(* IEC 61131-3 sources: elnaProjects/ElpcLogic/PomarKc7Changed/FunctionBlocks (part 7) *)

(* ---- proc_IM_Init.st ---- *)
FUNCTION_BLOCK proc_IM_Init

VAR_INPUT
	init : BOOL; (*Флаг необходимости инициализации структур-дескрипторов.*)
END_VAR

VAR
	stKr_Ini : fb_Kran_Init; (*ФБ инициализации кранов*)
	stSw_Ini : fb_Switch_Init; (*ФБ инициализации Switchs*)
	stOp_Ini : fb_OilPump_Init; (*ФБ инициализации НУ*)
	stSSw_Ini : fb_SectionSwitch_Init; (*ФБ инициализации МВ*)
	stAp_Ini : fb_AnalogParametr_Init; (*ФБ инициализации Аналогового параметра*)
	stDp_Ini : fb_DiscretParametr_Init; (*ФБ инициализации Дискретного параметра*)
	stSs_Ini : fb_singleSignal_Init; (*ФБ инициализации singleSignal*)
	stSo_Ini : fb_singleOutput_Init; (*ФБ инициализации singleOutput*)
	inits : UINT; (*Текущее количество успешно проинициализированных структур-дескрипторов.*)
END_VAR

VAR_INPUT
	initiales : UINT; (*Общее количество успешно проинициализированных структур-дескрипторов.*)
END_VAR

VAR_EXTERNAL
	IM : ImConfig;
END_VAR

inits := 0; (* Флаг необходимости инициализации структур-дескрипторов *)
                                     (* Стартовая инициализация ИМ *)
(* Кран 1 *)
stKr_Ini(data_Ini := true, ISVALIDREF_statOn:=true, ISVALIDREF_statOff:=true,
      ISVALIDREF_cmdOn:=true, ISVALIDREF_cmdOff:=true,
      ISVALIDREF_inSo:=true, ISVALIDREF_inSz:=true,
      str_Kr := IM.Kran1);
inits := inits + BOOL_TO_UINT(stKr_Ini.Init);

(* Кран 2 *)
stKr_Ini(data_Ini := true, ISVALIDREF_statOn:=true, ISVALIDREF_statOff:=true,
      ISVALIDREF_cmdOn:=true, ISVALIDREF_cmdOff:=true,
      ISVALIDREF_inSo:=true, ISVALIDREF_inSz:=true,
      str_Kr := IM.Kran2);
inits := inits + BOOL_TO_UINT(stKr_Ini.Init);

(* Кран 3 *)
stKr_Ini(data_Ini := true, ISVALIDREF_statOn:=true, ISVALIDREF_statOff:=true,
      ISVALIDREF_cmdOn:=true, ISVALIDREF_cmdOff:=true,
      ISVALIDREF_inSo:=true, ISVALIDREF_inSz:=true,
      str_Kr := IM.Kran3);
inits := inits + BOOL_TO_UINT(stKr_Ini.Init);

(* Кран 3b *)
stKr_Ini(data_Ini := true, ISVALIDREF_statOn:=true, ISVALIDREF_statOff:=true,
      ISVALIDREF_cmdOn:=true, ISVALIDREF_cmdOff:=true,
      ISVALIDREF_inSo:=true, ISVALIDREF_inSz:=true,
      str_Kr := IM.Kran3b);
inits := inits + BOOL_TO_UINT(stKr_Ini.Init);

(* Кран 4 *)
stKr_Ini(data_Ini := true, ISVALIDREF_statOn:=true, ISVALIDREF_statOff:=true,
      ISVALIDREF_cmdOn:=true, ISVALIDREF_cmdOff:=true,
      ISVALIDREF_inSo:=true, ISVALIDREF_inSz:=true,
      str_Kr := IM.Kran4);
inits := inits + BOOL_TO_UINT(stKr_Ini.Init);

(* Кран 5 *)
stKr_Ini(data_Ini := true, ISVALIDREF_statOn:=true, ISVALIDREF_statOff:=true,
      ISVALIDREF_cmdOn:=true, ISVALIDREF_cmdOff:=true,
      ISVALIDREF_inSo:=true, ISVALIDREF_inSz:=true, continueHoldCommand:=T#5S,
      str_Kr := IM.Kran5);
inits := inits + BOOL_TO_UINT(stKr_Ini.Init);

(* Кран 6 *)
stKr_Ini(data_Ini := true, ISVALIDREF_statOn:=true, ISVALIDREF_statOff:=true,
      ISVALIDREF_cmdOn:=true, ISVALIDREF_cmdOff:=true,
      str_Kr := IM.Kran6);
inits := inits + BOOL_TO_UINT(stKr_Ini.Init);

(* НУ1 Насос уплотнения *)
stOp_Ini(data_Ini := true, ISVALIDREF_statOn:=true, ISVALIDREF_statOff:=true,
      ISVALIDREF_cmdOn:=true, ISVALIDREF_cmdOff:=true,
      str_Op := IM.nu1);
inits := inits + BOOL_TO_UINT(stOp_Ini.Init);

(* НУ2 Насос уплотнения *)
stOp_Ini(data_Ini := true, ISVALIDREF_statOn:=true, ISVALIDREF_statOff:=true,
      ISVALIDREF_cmdOn:=true, ISVALIDREF_cmdOff:=true,
      str_Op := IM.nu2);
inits := inits + BOOL_TO_UINT(stOp_Ini.Init);

(* ПНС Насос смазки *)
stSw_Ini(data_Ini := true, ISVALIDREF_statOn:=true, ISVALIDREF_statOff:=true,
      ISVALIDREF_cmdOn:=true, ISVALIDREF_cmdOff:=true,
      str_Sw := IM.pns);
inits := inits + BOOL_TO_UINT(stSw_Ini.Init);

(* В1 АВОМ вентилятор охлаждения *)
stSw_Ini(data_Ini := true, ISVALIDREF_statOn:=true, ISVALIDREF_statOff:=true,
      ISVALIDREF_cmdOn:=true, ISVALIDREF_cmdOff:=true,
      str_Sw := IM.v1_Avom);
inits := inits + BOOL_TO_UINT(stSw_Ini.Init);

(* В2 АВОМ вентилятор охлаждения *)
stSw_Ini(data_Ini := true, ISVALIDREF_statOn:=true, ISVALIDREF_statOff:=true,
      ISVALIDREF_cmdOn:=true, ISVALIDREF_cmdOff:=true,
      str_Sw := IM.v2_Avom);
inits := inits + BOOL_TO_UINT(stSw_Ini.Init);

(* В3 АВОМ вентилятор охлаждения *)
stSw_Ini(data_Ini := true, ISVALIDREF_statOn:=true, ISVALIDREF_statOff:=true,
      ISVALIDREF_cmdOn:=true, ISVALIDREF_cmdOff:=true,
      str_Sw := IM.v3_Avom);
inits := inits + BOOL_TO_UINT(stSw_Ini.Init);

(* В4 АВОМ вентилятор охлаждения *)
stSw_Ini(data_Ini := true, ISVALIDREF_statOn:=true, ISVALIDREF_statOff:=true,
      ISVALIDREF_cmdOn:=true, ISVALIDREF_cmdOff:=true,
      str_Sw := IM.v4_Avom);
inits := inits + BOOL_TO_UINT(stSw_Ini.Init);

(* МВ масляный выключатель *)
stSSw_Ini(data_Ini := true, ISVALIDREF_statOn:=true, ISVALIDREF_statOff:=true,
      ISVALIDREF_cmdOn:=true, ISVALIDREF_cmdOff:=true,
      ISVALIDREF_basketRolledIn:=true, ISVALIDREF_basketRolledout:=true,
      str_Sw := IM.mv);
inits := inits + BOOL_TO_UINT(stSSw_Ini.Init);

(* В4 АВОМ вентилятор охлаждения *)
stSw_Ini(data_Ini := true, ISVALIDREF_statOn:=true, ISVALIDREF_statOff:=true,
      ISVALIDREF_cmdOn:=true, ISVALIDREF_cmdOff:=true,
      str_Sw := IM.KaloriferAVOM);
inits := inits + BOOL_TO_UINT(stSw_Ini.Init);

(* В4 АВОМ вентилятор охлаждения *)
stSw_Ini(data_Ini := true, ISVALIDREF_statOn:=true, ISVALIDREF_statOff:=true,
      ISVALIDREF_cmdOn:=true, ISVALIDREF_cmdOff:=true,
      str_Sw := IM.CMN);
inits := inits + BOOL_TO_UINT(stSw_Ini.Init);

(* В4 АВОМ вентилятор охлаждения *)
stSw_Ini(data_Ini := true, ISVALIDREF_statOn:=true, ISVALIDREF_statOff:=true,
      ISVALIDREF_cmdOn:=true, ISVALIDREF_cmdOff:=true,
      str_Sw := IM.TEN_kollectora);
inits := inits + BOOL_TO_UINT(stSw_Ini.Init);

(* В4 АВОМ вентилятор охлаждения *)
stSw_Ini(data_Ini := true, ISVALIDREF_statOn:=true, ISVALIDREF_statOff:=true,
      ISVALIDREF_cmdOn:=true, ISVALIDREF_cmdOff:=true,
      str_Sw := IM.TEN_MB);
inits := inits + BOOL_TO_UINT(stSw_Ini.Init);

                                     (* Стартовая инициализация singleSignal *)
    (* Перепад давления «газ-газ» на кране 1 ≤1 кгс/см² *)
stSs_Ini(data_Ini := true, inverse:=FALSE, (*DelayOn:=T#0S, DelayOff:=T#0S,*) str_SS := IM.SingleSignals.dP_maslo_gaz_Less100);
inits := inits + BOOL_TO_UINT(stSs_Ini.Init);

 (* Осевой сдвиг ротора вправо ≥3,7 кгс/см² *)
stSs_Ini(data_Ini := true, inverse:=FALSE, (*DelayOn:=T#0S, DelayOff:=T#0S,*) str_SS := IM.SingleSignals.dp_kran1_Less100);
inits := inits + BOOL_TO_UINT(stSs_Ini.Init);

    (* Пробой вентиля *)
stSs_Ini(data_Ini := true, inverse:=TRUE, (*DelayOn:=T#0S, DelayOff:=T#0S,*) str_SS := IM.SingleSignals.Vozbud_neispr_tsepey_upr_AVR_pit);
inits := inits + BOOL_TO_UINT(stSs_Ini.Init);

    (* Работа схемы ресинхронизации *)
stSs_Ini(data_Ini := true, inverse:=FALSE, (*DelayOn:=T#0S, DelayOff:=T#0S,*) str_SS := IM.SingleSignals.Vozbud_gotovnost);
inits := inits + BOOL_TO_UINT(stSs_Ini.Init);

    (* Контроль состояния возбудительного устройства  *)
stSs_Ini(data_Ini := true, inverse:=FALSE, (*DelayOn:=T#0S, DelayOff:=T#0S,*) str_SS := IM.SingleSignals.Vozbud_neispravnost);
inits := inits + BOOL_TO_UINT(stSs_Ini.Init);

    (* Неисправность форсировки воз-буждения  *)
stSs_Ini(data_Ini := true, inverse:=FALSE, (*DelayOn:=T#0S, DelayOff:=T#0S,*) str_SS := IM.SingleSignals.SHAVR1_v_rabote);
inits := inits + BOOL_TO_UINT(stSs_Ini.Init);

  (* Неисправность возбудительного устройства  *)
stSs_Ini(data_Ini := true, inverse:=FALSE, (*DelayOn:=T#0S, DelayOff:=T#0S,*) str_SS := IM.SingleSignals.SHAVR2_v_rabote);
inits := inits + BOOL_TO_UINT(stSs_Ini.Init);

  (* Готовность включения БЭО по отказу контроллера  *)
stSs_Ini(data_Ini := true, inverse:=FALSE, (*DelayOn:=T#0S, DelayOff:=T#0S,*) str_SS := IM.SingleSignals.Avariinoe_otkluch_vikluchatelya);
inits := inits + BOOL_TO_UINT(stSs_Ini.Init);

  (* Срабатывание БЭАО  *)
stSs_Ini(data_Ini := true, inverse:=FALSE, (*DelayOn:=T#0S, DelayOff:=T#0S,*) str_SS := IM.SingleSignals.Assinhronnii_hod_peregruzka);
inits := inits + BOOL_TO_UINT(stSs_Ini.Init);

  (* Выключатель основного ввода питания QF1  в положении включен   *)
stSs_Ini(data_Ini := true, inverse:=TRUE, (*DelayOn:=T#0S, DelayOff:=T#0S,*) str_SS := IM.SingleSignals.QF1_on);
inits := inits + BOOL_TO_UINT(stSs_Ini.Init);

  (* Выключатель резервного ввода питания QF2  в положении включен   *)
stSs_Ini(data_Ini := true, inverse:=TRUE, (*DelayOn:=T#0S, DelayOff:=T#0S,*) str_SS := IM.SingleSignals.QF2_on);
inits := inits + BOOL_TO_UINT(stSs_Ini.Init);

  (* Выключатель питания кранов:  QF23 110 В в положении включен   *)
stSs_Ini(data_Ini := true, inverse:=TRUE, (*DelayOn:=T#0S, DelayOff:=T#0S,*) str_SS := IM.SingleSignals.QF23_on);
inits := inits + BOOL_TO_UINT(stSs_Ini.Init);

  (* Выключатели группы 1: QF4, QF5 в положении включен   *)
stSs_Ini(data_Ini := true, inverse:=TRUE, (*DelayOn:=T#0S, DelayOff:=T#0S,*) str_SS := IM.SingleSignals.QF4_QF5_on);
inits := inits + BOOL_TO_UINT(stSs_Ini.Init);

  (* Выключатели группы 2: QF6, QF7 в положении включен   *)
stSs_Ini(data_Ini := true, inverse:=TRUE, (*DelayOn:=T#0S, DelayOff:=T#0S,*) str_SS := IM.SingleSignals.QF6_QF7_on);
inits := inits + BOOL_TO_UINT(stSs_Ini.Init);

  (* Выключатели группы 3: QF8, QF9 в положении включен   *)
stSs_Ini(data_Ini := true, inverse:=TRUE, (*DelayOn:=T#0S, DelayOff:=T#0S,*) str_SS := IM.SingleSignals.QF8_QF9_on);
inits := inits + BOOL_TO_UINT(stSs_Ini.Init);

  (* Выключатели группы 4: QF10, QF11 в положении включен   *)
stSs_Ini(data_Ini := true, inverse:=TRUE, (*DelayOn:=T#0S, DelayOff:=T#0S,*) str_SS := IM.SingleSignals.QF10_QF11_on);
inits := inits + BOOL_TO_UINT(stSs_Ini.Init);

  (* Выключатели группы 5: QF12, QF13 в положении включен   *)
stSs_Ini(data_Ini := true, inverse:=TRUE, (*DelayOn:=T#0S, DelayOff:=T#0S,*) str_SS := IM.SingleSignals.QF12_QF13_on);
inits := inits + BOOL_TO_UINT(stSs_Ini.Init);

  (* Выключатели группы 6: QF14, QF15 в положении включен   *)
stSs_Ini(data_Ini := true, inverse:=TRUE, (*DelayOn:=T#0S, DelayOff:=T#0S,*) str_SS := IM.SingleSignals.QF14_QF15_on);
inits := inits + BOOL_TO_UINT(stSs_Ini.Init);

  (* Выключатели группы : QF22 в положении включен   *)
stSs_Ini(data_Ini := true, inverse:=TRUE, (*DelayOn:=T#0S, DelayOff:=T#0S,*) str_SS := IM.SingleSignals.QF22_on);
inits := inits + BOOL_TO_UINT(stSs_Ini.Init);

  (* Неисправность источников питания группы 1: G1, G2 (=24 В)   *)
stSs_Ini(data_Ini := true, inverse:=TRUE, (*DelayOn:=T#0S, DelayOff:=T#0S,*) str_SS := IM.SingleSignals.NS_G1_G2);
inits := inits + BOOL_TO_UINT(stSs_Ini.Init);

  (* Неисправность источников питания группы 2: G3, G4 (=24 В)   *)
stSs_Ini(data_Ini := true, inverse:=TRUE, (*DelayOn:=T#0S, DelayOff:=T#0S,*) str_SS := IM.SingleSignals.NS_G3_G4);
inits := inits + BOOL_TO_UINT(stSs_Ini.Init);

  (* Неисправность источников питания внутренних ПТС: G15, G16 (=24 В)   *)
stSs_Ini(data_Ini := true, inverse:=TRUE, (*DelayOn:=T#0S, DelayOff:=T#0S,*) str_SS := IM.SingleSignals.NS_G15_G16);
inits := inits + BOOL_TO_UINT(stSs_Ini.Init);

  (* Неисправность источника питания аналоговых сигналов: G17 (=24 В)   *)
stSs_Ini(data_Ini := true, inverse:=TRUE, (*DelayOn:=T#0S, DelayOff:=T#0S,*) str_SS := IM.SingleSignals.NS_G17);
inits := inits + BOOL_TO_UINT(stSs_Ini.Init);

  (* Неисправность источников питания группы 3: G5, G6 (=24 В)   *)
stSs_Ini(data_Ini := true, inverse:=TRUE, (*DelayOn:=T#0S, DelayOff:=T#0S,*) str_SS := IM.SingleSignals.NS_G5_G6);
inits := inits + BOOL_TO_UINT(stSs_Ini.Init);

  (* Неисправность источников питания группы 4: G7, G8 (=24 В)   *)
stSs_Ini(data_Ini := true, inverse:=TRUE, (*DelayOn:=T#0S, DelayOff:=T#0S,*) str_SS := IM.SingleSignals.NS_G7_G8);
inits := inits + BOOL_TO_UINT(stSs_Ini.Init);

  (* Неисправность источников питания внешних цепей: G18, G19 (=24 В)   *)
stSs_Ini(data_Ini := true, inverse:=TRUE, (*DelayOn:=T#0S, DelayOff:=T#0S,*) str_SS := IM.SingleSignals.NS_G18_G19);
inits := inits + BOOL_TO_UINT(stSs_Ini.Init);

  (* Неисправность источников питания группы 5: G9, G10, G11, G12 (=110 В)   *)
stSs_Ini(data_Ini := true, inverse:=TRUE, (*DelayOn:=T#0S, DelayOff:=T#0S,*) str_SS := IM.SingleSignals.NS_G10_G11);
inits := inits + BOOL_TO_UINT(stSs_Ini.Init);

  (* Неисправность источников питания G13, G14 (=24 В)   *)
stSs_Ini(data_Ini := true, inverse:=TRUE, (*DelayOn:=T#0S, DelayOff:=T#0S,*) str_SS := IM.SingleSignals.NS_G13_G14);
inits := inits + BOOL_TO_UINT(stSs_Ini.Init);

    (* Неисправность источников питания G13, G14 (=24 В)   *)
stSs_Ini(data_Ini := true, inverse:=TRUE, (*DelayOn:=T#0S, DelayOff:=T#0S,*) str_SS := IM.SingleSignals.Uroven_masla_akkum);
inits := inits + BOOL_TO_UINT(stSs_Ini.Init);

  (* Неисправность источников питания G13, G14 (=24 В)   *)
stSs_Ini(data_Ini := true, inverse:=TRUE, (*DelayOn:=T#0S, DelayOff:=T#0S,*) str_SS := IM.SingleSignals.BEAO_srabotal);
inits := inits + BOOL_TO_UINT(stSs_Ini.Init);

  (* Неисправность источников питания G13, G14 (=24 В)   *)
stSs_Ini(data_Ini := true, inverse:=TRUE, (*DelayOn:=T#0S, DelayOff:=T#0S,*) str_SS := IM.SingleSignals.Chastotny_pusk);
inits := inits + BOOL_TO_UINT(stSs_Ini.Init);

  (* Неисправность источников питания G13, G14 (=24 В)   *)
stSs_Ini(data_Ini := true, inverse:=TRUE, (*DelayOn:=T#0S, DelayOff:=T#0S,*) str_SS := IM.SingleSignals.Neuspesh_chastotny_pusk);
inits := inits + BOOL_TO_UINT(stSs_Ini.Init);

  (* Неисправность источников питания G13, G14 (=24 В)   *)
stSs_Ini(data_Ini := true, inverse:=TRUE, (*DelayOn:=T#0S, DelayOff:=T#0S,*) str_SS := IM.SingleSignals.Rezhim_ruchnogo_regulirovaniya);
inits := inits + BOOL_TO_UINT(stSs_Ini.Init);

  (* Неисправность источников питания G13, G14 (=24 В)   *)
stSs_Ini(data_Ini := true, inverse:=TRUE, (*DelayOn:=T#0S, DelayOff:=T#0S,*) str_SS := IM.SingleSignals.SHU_v_GPA_vkluch);
inits := inits + BOOL_TO_UINT(stSs_Ini.Init);

  (* Неисправность источников питания G13, G14 (=24 В)   *)
stSs_Ini(data_Ini := true, inverse:=TRUE, (*DelayOn:=T#0S, DelayOff:=T#0S,*) str_SS := IM.SingleSignals.SHP_v_GPA_vkluch);
inits := inits + BOOL_TO_UINT(stSs_Ini.Init);

(* Отключение МВ1 от КНА   *)
stSs_Ini(data_Ini := true, inverse:=TRUE, (*wait_time:=T#0S,*) str_SS := IM.SingleSignals.NKU1_GPA_on);
inits := inits + BOOL_TO_UINT(stSs_Ini.Init);

(* Отключение МВ1 от КНА   *)
stSs_Ini(data_Ini := true, inverse:=TRUE, (*wait_time:=T#0S,*) str_SS := IM.SingleSignals.NKU2_GPA_on);
inits := inits + BOOL_TO_UINT(stSs_Ini.Init);

(* Отключение МВ1 от КНА   *)
stSs_Ini(data_Ini := true, inverse:=TRUE, (*wait_time:=T#0S,*) str_SS := IM.SingleSignals.AO_KC_ot_SHKS);
inits := inits + BOOL_TO_UINT(stSs_Ini.Init);

(* Отключение МВ1 от КНА   *)
stSs_Ini(data_Ini := true, inverse:=TRUE, (*wait_time:=T#0S,*) str_SS := IM.SingleSignals.AO_GPA_ot_SHU);
inits := inits + BOOL_TO_UINT(stSs_Ini.Init);

(* Отключение МВ1 от КНА   *)
stSs_Ini(data_Ini := true, inverse:=TRUE, (*wait_time:=T#0S,*) str_SS := IM.SingleSignals.Razreshenie_zagruzki_dvig);
inits := inits + BOOL_TO_UINT(stSs_Ini.Init);

(* Отключение МВ1 от КНА   *)
stSs_Ini(data_Ini := true, inverse:=TRUE, (*wait_time:=T#0S,*) str_SS := IM.SingleSignals.Osnovnoy_regul_off);
inits := inits + BOOL_TO_UINT(stSs_Ini.Init);

(* Отключение МВ1 от КНА   *)
stSs_Ini(data_Ini := true, inverse:=TRUE, (*wait_time:=T#0S,*) str_SS := IM.SingleSignals.Voltage_sekcii_norm);
inits := inits + BOOL_TO_UINT(stSs_Ini.Init);

(* Отключение МВ1 от КНА   *)
stSs_Ini(data_Ini := true, inverse:=TRUE, (*wait_time:=T#0S,*) str_SS := IM.SingleSignals.Reactorny_pusk);
inits := inits + BOOL_TO_UINT(stSs_Ini.Init);

(* Отключение МВ1 от КНА   *)
stSs_Ini(data_Ini := true, inverse:=TRUE, (*wait_time:=T#0S,*) str_SS := IM.SingleSignals.NO_GPA_ot_SHU);
inits := inits + BOOL_TO_UINT(stSs_Ini.Init);

(* Отключение МВ1 от КНА   *)
stSs_Ini(data_Ini := true, inverse:=TRUE, (*wait_time:=T#0S,*) str_SS := IM.SingleSignals.AO_GPA_ot_PRU);
inits := inits + BOOL_TO_UINT(stSs_Ini.Init);

(* Отключение МВ1 от КНА   *)
stSs_Ini(data_Ini := true, inverse:=TRUE, (*wait_time:=T#0S,*) str_SS := IM.SingleSignals.Nalichie_BP1);
inits := inits + BOOL_TO_UINT(stSs_Ini.Init);

(* Отключение МВ1 от КНА   *)
stSs_Ini(data_Ini := true, inverse:=TRUE, (*wait_time:=T#0S,*) str_SS := IM.SingleSignals.Nalichie_BP2);
inits := inits + BOOL_TO_UINT(stSs_Ini.Init);

(* Отключение МВ1 от КНА   *)
stSs_Ini(data_Ini := true, inverse:=TRUE, (*wait_time:=T#0S,*) str_SS := IM.SingleSignals.Nalichie_BP3);
inits := inits + BOOL_TO_UINT(stSs_Ini.Init);

(* Отключение МВ1 от КНА   *)
stSs_Ini(data_Ini := true, inverse:=TRUE, (*wait_time:=T#0S,*) str_SS := IM.SingleSignals.Nalichie_BP4);
inits := inits + BOOL_TO_UINT(stSs_Ini.Init);

(* Отключение МВ1 от КНА   *)
stSs_Ini(data_Ini := true, inverse:=TRUE, (*wait_time:=T#0S,*) str_SS := IM.SingleSignals.Nalichie_BP5);
inits := inits + BOOL_TO_UINT(stSs_Ini.Init);

(* Отключение МВ1 от КНА   *)
stSs_Ini(data_Ini := true, inverse:=TRUE, (*wait_time:=T#0S,*) str_SS := IM.SingleSignals.Nalichie_BP6);
inits := inits + BOOL_TO_UINT(stSs_Ini.Init);

(* Отключение МВ1 от КНА   *)
stSs_Ini(data_Ini := true, inverse:=TRUE, (*wait_time:=T#0S,*) str_SS := IM.SingleSignals.Nalichie_BP7_BP8);
inits := inits + BOOL_TO_UINT(stSs_Ini.Init);

(* Отключение МВ1 от КНА   *)
stSs_Ini(data_Ini := true, inverse:=TRUE, (*wait_time:=T#0S,*) str_SS := IM.SingleSignals.Nalichie_BP9_BP10);
inits := inits + BOOL_TO_UINT(stSs_Ini.Init);

(* Отключение МВ1 от КНА   *)
stSs_Ini(data_Ini := true, inverse:=TRUE, (*wait_time:=T#0S,*) str_SS := IM.SingleSignals.Nalichie_cepei_upravlen_mv);
inits := inits + BOOL_TO_UINT(stSs_Ini.Init);

(* Отключение МВ1 от КНА   *)
stSs_Ini(data_Ini := true, inverse:=TRUE, (*wait_time:=T#0S,*) str_SS := IM.SingleSignals.Nalichie_220BEAO);
inits := inits + BOOL_TO_UINT(stSs_Ini.Init);

(* Отключение МВ1 от КНА   *)
stSs_Ini(data_Ini := true, inverse:=TRUE, (*wait_time:=T#0S,*) str_SS := IM.SingleSignals.Nalichie_per_220_na_vhode);
inits := inits + BOOL_TO_UINT(stSs_Ini.Init);

(* Отключение МВ1 от КНА   *)
stSs_Ini(data_Ini := true, inverse:=TRUE, (*wait_time:=T#0S,*) str_SS := IM.SingleSignals.Nalichie_post_220_na_vhode);
inits := inits + BOOL_TO_UINT(stSs_Ini.Init);

(* Отключение МВ1 от КНА   *)
stSs_Ini(data_Ini := true, inverse:=TRUE, (*wait_time:=T#0S,*) str_SS := IM.SingleSignals.Nalichie_BP11);
inits := inits + BOOL_TO_UINT(stSs_Ini.Init);

(* Отключение МВ1 от КНА   *)
stSs_Ini(data_Ini := true, inverse:=TRUE, (*wait_time:=T#0S,*) str_SS := IM.SingleSignals.Nalichie_BP12);
inits := inits + BOOL_TO_UINT(stSs_Ini.Init);

(* Отключение МВ1 от КНА   *)
stSs_Ini(data_Ini := true, inverse:=TRUE, (*wait_time:=T#0S,*) str_SS := IM.SingleSignals.Dver_SHU_pered_otkrita);
inits := inits + BOOL_TO_UINT(stSs_Ini.Init);

(* Отключение МВ1 от КНА   *)
stSs_Ini(data_Ini := true, inverse:=TRUE, (*wait_time:=T#0S,*) str_SS := IM.SingleSignals.Dver_SHU_zad_otkrita);
inits := inits + BOOL_TO_UINT(stSs_Ini.Init);

(* Отключение МВ1 от КНА   *)
stSs_Ini(data_Ini := true, inverse:=TRUE, (*wait_time:=T#0S,*) str_SS := IM.SingleSignals.EO_GPA_ot_knopki_SHU);
inits := inits + BOOL_TO_UINT(stSs_Ini.Init);

(* Отключение МВ1 от КНА   *)
stSs_Ini(data_Ini := true, inverse:=TRUE, (*wait_time:=T#0S,*) str_SS := IM.SingleSignals.EO_EGPA_ot_PRY);
inits := inits + BOOL_TO_UINT(stSs_Ini.Init);

(* Отключение МВ1 от КНА   *)
stSs_Ini(data_Ini := true, inverse:=TRUE, (*wait_time:=T#0S,*) str_SS := IM.SingleSignals.Synchroniz_rezhima_K1);
inits := inits + BOOL_TO_UINT(stSs_Ini.Init);

                                     (* Стартовая инициализация singleOutput *)
(* Идикация НО (подсветка кнопки на шкафу)   *)
stSo_Ini(data_Ini := true, inOpcCommandsDisabled:=TRUE, (*wait_time:=T#0S,*) str_SO := IM.SingleOutputs.Rabota_EGPA);
inits := inits + BOOL_TO_UINT(stSo_Ini.Init);

(* Взвод включения БЭАО по неисправности ПТС   *)
stSo_Ini(data_Ini := true, inOpcCommandsDisabled:=TRUE, wait_time:=T#0S, str_SO := IM.SingleOutputs.Neispr_EGPA);
inits := inits + BOOL_TO_UINT(stSo_Ini.Init);

(* Авария ЭГПА в КЦ   *)
stSo_Ini(data_Ini := true, inOpcCommandsDisabled:=TRUE, (*wait_time:=T#0S,*) str_SO := IM.SingleOutputs.Avary_EGPA);
inits := inits + BOOL_TO_UINT(stSo_Ini.Init);

(* Авария ЭГПА в КЦ   *)
stSo_Ini(data_Ini := true, inOpcCommandsDisabled:=TRUE, (*wait_time:=T#0S,*) str_SO := IM.SingleOutputs.U_lamp_SHU);
inits := inits + BOOL_TO_UINT(stSo_Ini.Init);

(* Индикация ПС Фонарь   *)
stSo_Ini(data_Ini := true, inOpcCommandsDisabled:=TRUE, (*wait_time:=T#0S,*) str_SO := IM.SingleOutputs.AO_knopka_ind);
inits := inits + BOOL_TO_UINT(stSo_Ini.Init);

(* Индикация АС Фонарь   *)
stSo_Ini(data_Ini := true, inOpcCommandsDisabled:=TRUE, (*wait_time:=T#0S,*) str_SO := IM.SingleOutputs.Pusk_SHUP);
inits := inits + BOOL_TO_UINT(stSo_Ini.Init);

(* Отключение МВ1 от КНА   *)
stSo_Ini(data_Ini := true, inOpcCommandsDisabled:=TRUE, (*wait_time:=T#0S,*) str_SO := IM.SingleOutputs.Stop_SHUP);
inits := inits + BOOL_TO_UINT(stSo_Ini.Init);

(* Отключение МВ1 от КНА   *)
stSo_Ini(data_Ini := true, inOpcCommandsDisabled:=TRUE, (*wait_time:=T#0S,*) str_SO := IM.SingleOutputs.NO_fonar);
inits := inits + BOOL_TO_UINT(stSo_Ini.Init);

(* Отключение МВ1 от КНА   *)
stSo_Ini(data_Ini := true, inOpcCommandsDisabled:=TRUE, (*wait_time:=T#0S,*) str_SO := IM.SingleOutputs.PC_fonar);
inits := inits + BOOL_TO_UINT(stSo_Ini.Init);

(* Отключение МВ1 от КНА   *)
stSo_Ini(data_Ini := true, inOpcCommandsDisabled:=TRUE, (*wait_time:=T#0S,*) str_SO := IM.SingleOutputs.AC_fonar);
inits := inits + BOOL_TO_UINT(stSo_Ini.Init);

(* Отключение МВ1 от КНА   *)
stSo_Ini(data_Ini := true, inOpcCommandsDisabled:=TRUE, (*wait_time:=T#0S,*) str_SO := IM.SingleOutputs.Kr1_smazka);
inits := inits + BOOL_TO_UINT(stSo_Ini.Init);

(* Отключение МВ1 от КНА   *)
stSo_Ini(data_Ini := true, inOpcCommandsDisabled:=TRUE, (*wait_time:=T#0S,*) str_SO := IM.SingleOutputs.Kr2_smazka);
inits := inits + BOOL_TO_UINT(stSo_Ini.Init);

(* Отключение МВ1 от КНА   *)
stSo_Ini(data_Ini := true, inOpcCommandsDisabled:=TRUE, (*wait_time:=T#0S,*) str_SO := IM.SingleOutputs.Kr4_open_from_alg);
inits := inits + BOOL_TO_UINT(stSo_Ini.Init);

(* Отключение МВ1 от КНА   *)
stSo_Ini(data_Ini := true, inOpcCommandsDisabled:=TRUE, (*wait_time:=T#0S,*) str_SO := IM.SingleOutputs.Synch_rej_K1);
inits := inits + BOOL_TO_UINT(stSo_Ini.Init);
initiales := 0;

IF init THEN initiales := inits; END_IF;

(* ---- proc_Protection.st ---- *)
FUNCTION_BLOCK proc_Protection

VAR
	fb_mvOff : fb_MvProtection;
	fb_dPmaslo_gaz_Less100 : fb_DiProtection; (*[A1-14:1, AI0] Резерв*)
	fb_Reg_vozb_off : fb_DiProtection; (*[A1-14:2, AI1] Резерв*)
	fb_Fail_chastotnii_pusk : fb_DiProtection;
	fb_Off_avar_vikluchatel : fb_DiProtection;
	fb_AOKC_SHKC : fb_DiProtection;
	fb_AO_PRU : fb_DiProtection;
	fb_AO_ot_SHU : fb_DiProtection;
	fb_Kran1_sdvig : fb_KranOpenProtection;
	fb_Kran2_sdvig : fb_KranOpenProtection;
	fb_Toporno_podshipnika_EDT_1 : fb_AiProtection;
	fb_Toy_podshipnika_EDT_2 : fb_AiProtection;
	fb_Toy_podshipnika_kol_EDT_3 : fb_AiProtection;
	fb_Toy_podshipnika_kol_EDT_4 : fb_AiProtection;
	fb_Toy_podshipnika_shest_red_EDT_5 : fb_AiProtection;
	fb_Ty_podshipnika_red_EDT_6 : fb_AiProtection;
	fb_Ty_podshipnika_nagnet_EDT_7_1 : fb_AiProtection;
	fb_Ty_podshipnika_nagnet_EDT_7_2 : fb_AiProtection;
	fb_Toy_podshipnika_svobod_konca_EDT_8_1 : fb_AiProtection;
	fb_Toy_podshipnika_svobod_konca_EDT_8_2 : fb_AiProtection;
	fb_Toy_podshipnika_rab_kol_EDT_9_1 : fb_AiProtection;
	fb_Toy_podshipnika_rab_kol_EDT_9_2 : fb_AiProtection;
	fb_Toy_podshipnika_nerab_kol_EDT_10_1 : fb_AiProtection;
	fb_Toy_podshipnika_nerab_kol_EDT_10_2 : fb_AiProtection;
	fb_Tgaza_na_vhode_H : fb_AiProtection;
	fb_Tgaza_na_vyhode_H : fb_AiProtection;
	fb_Tmasla_v_mb : fb_AiProtection;
	fb_Tmasla_v_mb_nad_ten : fb_AiProtection;
	fb_Tgorjachego_vozduha_ED_kanal_1 : fb_AiProtection;
	fb_Tgorjachego_vozduha_ED_kanal_2 : fb_AiProtection;
	fb_Tmasla_do_AVOM : fb_AiProtection;
	fb_Tmasla_posle_AVOM : fb_AiProtection;
	fb_Tmedi_statora_kanal_1 : fb_AiProtection;
	fb_Tmedi_statora_kanal_2 : fb_AiProtection;
	fb_Tmedi_statora_kanal_3 : fb_AiProtection;
	fb_Tstali_statora_kanal_1 : fb_AiProtection;
	fb_Tstali_statora_kanal_2 : fb_AiProtection;
	fb_Tstali_statora_kanal_3 : fb_AiProtection;
	fb_Tholodnogo_vozduha_ED_kanal_1 : fb_AiProtection;
	fb_Tholodnogo_vozduha_ED_kanal_2 : fb_AiProtection;
	fb_Pmaslo_sm_nizkoe : fb_AiProtection;
	fb_Pmaslo_sm_vysokoe : fb_AiProtection;
	fb_Pgaza_na_vhode_nagnetatelia : fb_AiProtection;
	fb_Pgaza_na_vyhode_nagnetatelia : fb_AiProtection;
	fb_Pmasla_posle_NU : fb_AiProtection;
	fb_Pmasla_smazki_posle_gns : fb_AiProtection;
	fb_Pimpuls_gaz : fb_AiProtection;
	fb_dPmaslo_gaz : fb_AiProtection;
	fb_dP_maslo_na_filtre : fb_AiProtection;
	fb_Os_sdvig_nagnetatelja_plus : fb_AiProtection;
	fb_Os_sdvig_nagnetatelja_minus : fb_AiProtection;
	fb_Vibro_skorost_OPED_T1 : fb_AiProtection;
	fb_Vibro_skorost_OPED_T2 : fb_AiProtection;
	fb_Vibro_skorost_OYP_kolesa_ED_T3 : fb_AiProtection;
	fb_Vibro_skorost_OP_kolesa_RH_T4 : fb_AiProtection;
	fb_Vibro_skorost_OP_shesterni_RED_T5 : fb_AiProtection;
	fb_Vibro_skorost_OP_shesterni_RED_T6 : fb_AiProtection;
	fb_Vibroperemesh_vala_N_T7 : fb_AiProtection;
	fb_Vibroperemesh_vala_N_T8 : fb_AiProtection;
	fb_Uroven_masla_v_mb : fb_AiProtection;
	fb_Tok_statora : fb_AiProtection;
	fb_Kontrol_per_220V_less187 : fb_AiProtection;
	fb_Kontrol_per_220V_high242 : fb_AiProtection;
	fb_Kontrol_post_220V_less187 : fb_AiProtection;
	fb_Kontrol_post_220V_high242 : fb_AiProtection;
END_VAR

VAR_EXTERNAL
	protections : ProtectionsConfig;
	ai : AiConfig;
	IM : ImConfig;
END_VAR

(************************************************************* DiProtection ************************************************************)
(* МВ отключен
fb_mvOff(sw:=IM.mv, StrDIp := protections.Pgaza_na_vyhode_nagnetatelia_GPA_STOP);*)

(* Неисправность возбудительного устройства *)
fb_dPmaslo_gaz_Less100(di := IM.SingleSignals.dP_maslo_gaz_Less100, StrDIp := protections.dPmaslo_gaz_less100);

(* Сдвиг крана №2 *)
fb_Reg_vozb_off(di:=IM.SingleSignals.Vozbud_neispravnost, StrDIp := protections.Reg_vozb_off);

(* Сдвиг крана №2 *)
fb_Fail_chastotnii_pusk(di:=IM.SingleSignals.Neuspesh_chastotny_pusk, StrDIp := protections.Fail_chastotnii_pusk);

(* Сдвиг крана №2 *)
fb_Off_avar_vikluchatel(di:=IM.SingleSignals.Avariinoe_otkluch_vikluchatelya, StrDIp := protections.Off_avar_vikluchatel);

(* Сдвиг крана №2 *)
fb_AOKC_SHKC(di:=IM.SingleSignals.AO_KC_ot_SHKS, StrDIp := protections.AOKC_SHKC);

(* Сдвиг крана №2 *)
fb_AO_PRU(di:=IM.SingleSignals.AO_GPA_ot_PRU, StrDIp := protections.AO_PRU);

(* Сдвиг крана №2 *)
fb_AO_ot_SHU(di:=IM.SingleSignals.AO_GPA_ot_SHU, StrDIp := protections.AO_ot_SHU);

(* Сдвиг крана №2 *)
fb_Kran1_sdvig(im:=IM.Kran1, StrDIp := protections.Kran1_sdvig);

(* Сдвиг крана №2 *)
fb_Kran2_sdvig(im:=IM.Kran2, StrDIp := protections.Kran2_sdvig);

(************************************************************* AiProtection ************************************************************)

(* Температура переднего опорного подшипника двигателя, т.1 *)
fb_Toporno_podshipnika_EDT_1(ai := ai.Toporno_podshipnika_EDT_1, StrAIp := protections.Topornogo_podshipnika_EDT_1);

(* Температура заднего опорного подшипника двигателя, т.2 *)
fb_Toy_podshipnika_EDT_2(ai := ai.Toy_podshipnika_EDT_2, StrAIp := protections.Toy_podshipnika_EDT_2);

(* Температура подшипника редуктора, т1 *)
fb_Toy_podshipnika_kol_EDT_3(ai := ai.Toy_podshipnika_kol_EDT_3, StrAIp := protections.Toy_podshipnika_kol_EDT_3);

(* Температура подшипника редуктора, т2 *)
fb_Toy_podshipnika_kol_EDT_4(ai := ai.Toy_podshipnika_kol_EDT_4, StrAIp := protections.Toy_podshipnika_kol_EDT_4);

(* Температура подшипника редуктора, т3 *)
fb_Toy_podshipnika_shest_red_EDT_5(ai := ai.Toy_podshipnika_shest_red_EDT_5, StrAIp := protections.To_podshipnika_shest_red_EDT_5);

(* Температура подшипника редуктора, т4 *)
fb_Ty_podshipnika_red_EDT_6(ai := ai.Ty_podshipnika_red_EDT_6, StrAIp := protections.To_podshipnika_shest_red_EDT_6);

(* Температура опорного подшипника нагнетателя, т1 *)
fb_Ty_podshipnika_nagnet_EDT_7_1(ai := ai.Ty_podshipnika_nagnet_EDT_7_1, StrAIp := protections.To_podshipnika_N_EDT_7);

(* Температура опорного подшипника нагнетателя, т1 *)
fb_Ty_podshipnika_nagnet_EDT_7_2(ai := ai.Ty_podshipnika_nagnet_EDT_7_2, StrAIp := protections.To_podshipnika_N_EDT_7);

(* Температура опорного подшипника нагнетателя, т2 *)
fb_Toy_podshipnika_svobod_konca_EDT_8_1(ai := ai.Toy_podshipnika_svobod_konca_EDT_8_1, StrAIp := protections.To_podshipnika_svob_konca_EDT_8);

(* Температура опорного подшипника нагнетателя, т2 *)
fb_Toy_podshipnika_svobod_konca_EDT_8_2(ai := ai.Toy_podshipnika_svobod_konca_EDT_8_2, StrAIp := protections.To_podshipnika_svob_konca_EDT_8);

(* Температура опорного подшипника нагнетателя, т3 *)
fb_Toy_podshipnika_rab_kol_EDT_9_1(ai := ai.Toy_podshipnika_rab_kol_EDT_9_1, StrAIp := protections.Ty_podshipnika_rab_kol_EDT_9);

(* Температура опорного подшипника нагнетателя, т3 *)
fb_Toy_podshipnika_rab_kol_EDT_9_2(ai := ai.Toy_podshipnika_rab_kol_EDT_9_2, StrAIp := protections.Ty_podshipnika_rab_kol_EDT_9);

(* Температура упорно опорного подшипника нагнетателя, т4 *)
fb_Toy_podshipnika_nerab_kol_EDT_10_1(ai := ai.Toy_podshipnika_nerab_kol_EDT_10_1, StrAIp := protections.Typornogo_podshipnika_nerab_kolodok_HT_10);

(* Температура упорно опорного подшипника нагнетателя, т4 *)
fb_Toy_podshipnika_nerab_kol_EDT_10_2(ai := ai.Toy_podshipnika_nerab_kol_EDT_10_2, StrAIp := protections.Typornogo_podshipnika_nerab_kolodok_HT_10);

(* Температура газа на выходе нагнетателя *)
fb_Tgaza_na_vyhode_H(ai := ai.Tgaza_na_vhode_H, StrAIp := protections.Tgaza_na_vyhode_H);

(* Температура газа на выходе нагнетателя *)
fb_Os_sdvig_nagnetatelja_plus(ai := ai.Os_sdvig_nagnetatelja_plus, StrAIp := protections.Os_sdvig_nagnetatelja_plus);

(* Температура газа на выходе нагнетателя *)
fb_Os_sdvig_nagnetatelja_minus(ai := ai.Os_sdvig_nagnetatelja_minus, StrAIp := protections.Os_sdvig_nagnetatelja_minus);

(* Температура газа на выходе нагнетателя *)
fb_Pgaza_na_vyhode_nagnetatelia(ai := ai.Pgaza_na_vyhode_nagnetatelia, StrAIp := protections.Pgaza_na_vyhode_nagnetatelia);

(* Температура газа на выходе нагнетателя *)
fb_dPmaslo_gaz(ai := ai.dPmaslo_gaz, StrAIp := protections.dPmaslo_gaz);

(* Температура газа на выходе нагнетателя *)
fb_Pmaslo_sm_nizkoe(ai := ai.Pmaslo_sm_nizkoe, StrAIp := protections.Pmaslo_sm_nizkoe);

(* Температура газа на выходе нагнетателя *)
fb_Pmaslo_sm_vysokoe(ai := ai.Pmaslo_sm_vysokoe, StrAIp := protections.Pmaslo_sm_vysokoe);

(* Температура газа на выходе нагнетателя *)
fb_Vibro_skorost_OPED_T1(ai := ai.Vibro_skorost_OPED_T1, StrAIp := protections.Vibro_skorost_OPED_T1);

(* Температура газа на выходе нагнетателя *)
fb_Vibro_skorost_OPED_T2(ai := ai.Vibro_skorost_OYPED_T2, StrAIp := protections.Vibro_skorost_OPED_T2);

(* Температура газа на выходе нагнетателя *)
fb_Vibro_skorost_OYP_kolesa_ED_T3(ai := ai.Vibro_skorost_OYP_kolesa_ED_T3, StrAIp := protections.Vibro_skorost_OYP_kolesa_ED_T3);

(* Температура газа на выходе нагнетателя *)
fb_Vibro_skorost_OP_kolesa_RH_T4(ai := ai.Vibro_skorost_OP_kolesa_RH_T4, StrAIp := protections.Vibro_skorost_OP_kolesa_RH_T4);

(* Температура газа на выходе нагнетателя *)
fb_Vibro_skorost_OP_shesterni_RED_T5(ai := ai.Vibro_skorost_OP_shesterni_RED_T5, StrAIp := protections.Vibro_skorost_OP_shesterni_RED_T5);

(* Температура газа на выходе нагнетателя *)
fb_Vibro_skorost_OP_shesterni_RED_T6(ai := ai.Vibro_skorost_OP_shesterni_RED_T6, StrAIp := protections.Vibro_skorost_OP_shesterni_RED_T6);

(* ---- proc_Protections_Init.st ---- *)
FUNCTION_BLOCK proc_Protections_Init

VAR_INPUT
	init : BOOL; (*Флаг необходимости инициализации структур-дескрипторов.*)
END_VAR

VAR
	stDIp_Ini : fb_DiProtection_Init; (*ФБ инициализации DiProtection*)
	stAIp_Ini : fb_AiProtection_Init; (*ФБ инициализации AiProtection*)
	inits : UINT; (*Текущее количество успешно проинициализированных структур-дескрипторов.*)
END_VAR

VAR_INPUT
	initiales : UINT; (*Общее количество успешно проинициализированных структур-дескрипторов.*)
END_VAR

VAR_EXTERNAL
	protections : ProtectionsConfig;
END_VAR

VAR
	_ProtectionTags : TYPE_ProtectionTags;
	_StatusAi : TYPE_StatusAi;
END_VAR

inits := 0; (* Флаг необходимости инициализации структур-дескрипторов *)

(*************************************************Стартовая инициализация DiProtection ***************************************************)
(* МВ отключен *)
stDIp_Ini(data_Ini := true, delay:=T#03S, inTag:=_ProtectionTags.AOS, inRunOnStart:=TRUE, str_DIp := protections.Reg_vozb_off);
inits := inits + BOOL_TO_UINT(stDIp_Ini.Init);

(* МВ отключен
stDIp_Ini(data_Ini := true, delay:=T#1S, inTag:=_ProtectionTags.AOS, inRunOnStart:=FALSE, str_DIp := protections.Fail_chastotnii_pusk);
inits := inits + BOOL_TO_UINT(stDIp_Ini.Init);*)

(* МВ отключен *)
stDIp_Ini(data_Ini := true, delay:=T#1S, inTag:=_ProtectionTags.AOS, inRunOnStart:=TRUE, str_DIp := protections.Off_avar_vikluchatel);
inits := inits + BOOL_TO_UINT(stDIp_Ini.Init);

(* МВ отключен *)
stDIp_Ini(data_Ini := true, delay:=T#1S, inTag:=_ProtectionTags.AOS, inRunOnStart:=TRUE, str_DIp := protections.AOKC_SHKC);
inits := inits + BOOL_TO_UINT(stDIp_Ini.Init);

(* МВ отключен *)
stDIp_Ini(data_Ini := true, delay:=T#0S, inTag:=_ProtectionTags.AOS, inRunOnStart:=TRUE, str_DIp := protections.AO_PRU);
inits := inits + BOOL_TO_UINT(stDIp_Ini.Init);

(* МВ отключен *)
stDIp_Ini(data_Ini := true, delay:=T#0S, inTag:=_ProtectionTags.AOS, inRunOnStart:=FALSE, str_DIp := protections.AO_ot_SHU);
inits := inits + BOOL_TO_UINT(stDIp_Ini.Init);

(* МВ отключен *)
stDIp_Ini(data_Ini := true, delay:=T#1S, inTag:=_ProtectionTags.AOS, inRunOnStart:=FALSE, str_DIp := protections.mvOff);
inits := inits + BOOL_TO_UINT(stDIp_Ini.Init);

(* МВ отключен *)
stDIp_Ini(data_Ini := true, delay:=T#10S, inTag:=_ProtectionTags.AOS, inRunOnStart:=TRUE, str_DIp := protections.Kran1_sdvig);
inits := inits + BOOL_TO_UINT(stDIp_Ini.Init);

(* МВ отключен *)
stDIp_Ini(data_Ini := true, delay:=T#10S, inTag:=_ProtectionTags.AOS, inRunOnStart:=TRUE, str_DIp := protections.Kran2_sdvig);
inits := inits + BOOL_TO_UINT(stDIp_Ini.Init);

(* МВ отключен *)
stDIp_Ini(data_Ini := true, delay:=T#20S, inTag:=_ProtectionTags.AOS, inRunOnStart:=TRUE, str_DIp := protections.dPmaslo_gaz_less100);
inits := inits + BOOL_TO_UINT(stDIp_Ini.Init);

(*************************************************Стартовая инициализация AiProtection ***************************************************)
(* Температура переднего опорного подшипника двигателя, т.1 *)
stAIp_Ini(data_Ini := true, delay:=T#3S, inTag:=_ProtectionTags.AOS, inRunOnStart:=TRUE,
controlLimit:=_StatusAi.HA, str_AIp := protections.Topornogo_podshipnika_EDT_1);
inits := inits + BOOL_TO_UINT(stAIp_Ini.Init);

(* Температура заднего опорного подшипника двигателя, т.2 *)
stAIp_Ini(data_Ini := true, delay:=T#3S, inTag:=_ProtectionTags.AOS, inRunOnStart:=TRUE,
controlLimit:=_StatusAi.HA, str_AIp := protections.Toy_podshipnika_EDT_2);
inits := inits + BOOL_TO_UINT(stAIp_Ini.Init);

(* Температура подшипника редуктора, т1 *)
stAIp_Ini(data_Ini := true, delay:=T#3S, inTag:=_ProtectionTags.AOS, inRunOnStart:=TRUE,
controlLimit:=_StatusAi.HA, str_AIp := protections.Toy_podshipnika_kol_EDT_3);
inits := inits + BOOL_TO_UINT(stAIp_Ini.Init);

(* Температура подшипника редуктора, т2 *)
stAIp_Ini(data_Ini := true, delay:=T#3S, inTag:=_ProtectionTags.AOS, inRunOnStart:=TRUE,
controlLimit:=_StatusAi.HA, str_AIp := protections.Toy_podshipnika_kol_EDT_4);
inits := inits + BOOL_TO_UINT(stAIp_Ini.Init);

(* Температура подшипника редуктора, т3 *)
stAIp_Ini(data_Ini := true, delay:=T#3S, inTag:=_ProtectionTags.AOS, inRunOnStart:=TRUE,
controlLimit:=_StatusAi.HA, str_AIp := protections.To_podshipnika_shest_red_EDT_5);
inits := inits + BOOL_TO_UINT(stAIp_Ini.Init);

(* Температура подшипника редуктора, т4 *)
stAIp_Ini(data_Ini := true, delay:=T#3S, inTag:=_ProtectionTags.AOS, inRunOnStart:=TRUE,
controlLimit:=_StatusAi.HA, str_AIp := protections.To_podshipnika_shest_red_EDT_6);
inits := inits + BOOL_TO_UINT(stAIp_Ini.Init);

(* Температура опорного подшипника нагнетателя, т1 *)
stAIp_Ini(data_Ini := true, delay:=T#3S, inTag:=_ProtectionTags.AOS, inRunOnStart:=TRUE,
controlLimit:=_StatusAi.HA, str_AIp := protections.To_podshipnika_N_EDT_7);
inits := inits + BOOL_TO_UINT(stAIp_Ini.Init);

(* Температура опорного подшипника нагнетателя, т2 *)
stAIp_Ini(data_Ini := true, delay:=T#3S, inTag:=_ProtectionTags.AOS, inRunOnStart:=TRUE,
controlLimit:=_StatusAi.HA, str_AIp := protections.To_podshipnika_svob_konca_EDT_8);
inits := inits + BOOL_TO_UINT(stAIp_Ini.Init);

(* Температура опорного подшипника нагнетателя, т3 *)
stAIp_Ini(data_Ini := true, delay:=T#3S, inTag:=_ProtectionTags.AOS, inRunOnStart:=TRUE,
controlLimit:=_StatusAi.HA, str_AIp := protections.Ty_podshipnika_rab_kol_EDT_9);
inits := inits + BOOL_TO_UINT(stAIp_Ini.Init);

(* Температура упорно опорного подшипника нагнетателя, т4 *)
stAIp_Ini(data_Ini := true, delay:=T#3S, inTag:=_ProtectionTags.AOS, inRunOnStart:=TRUE,
controlLimit:=_StatusAi.HA, str_AIp := protections.Typornogo_podshipnika_nerab_kolodok_HT_10);
inits := inits + BOOL_TO_UINT(stAIp_Ini.Init);

(* Температура газа на выходе нагнетателя *)
stAIp_Ini(data_Ini := true, delay:=T#3S, inTag:=_ProtectionTags.AOS, inRunOnStart:=TRUE,
controlLimit:=_StatusAi.HA, str_AIp := protections.Tgaza_na_vyhode_H);
inits := inits + BOOL_TO_UINT(stAIp_Ini.Init);

(* Температура газа на выходе нагнетателя *)
stAIp_Ini(data_Ini := true, delay:=T#3S, inTag:=_ProtectionTags.AOS, inRunOnStart:=TRUE,
controlLimit:=_StatusAi.HA, str_AIp := protections.Os_sdvig_nagnetatelja_plus);
inits := inits + BOOL_TO_UINT(stAIp_Ini.Init);

(* Температура газа на выходе нагнетателя *)
stAIp_Ini(data_Ini := true, delay:=T#3S, inTag:=_ProtectionTags.AOS, inRunOnStart:=TRUE,
controlLimit:=_StatusAi.HA, str_AIp := protections.Os_sdvig_nagnetatelja_minus);
inits := inits + BOOL_TO_UINT(stAIp_Ini.Init);

(* Температура газа на выходе нагнетателя *)
stAIp_Ini(data_Ini := true, delay:=T#3S, inTag:=_ProtectionTags.AOS, inRunOnStart:=TRUE,
controlLimit:=_StatusAi.HA, str_AIp := protections.Pgaza_na_vyhode_nagnetatelia_GPA_STOP);
inits := inits + BOOL_TO_UINT(stAIp_Ini.Init);

(* Температура газа на выходе нагнетателя *)
stAIp_Ini(data_Ini := true, delay:=T#3S, inTag:=_ProtectionTags.AOS, inRunOnStart:=TRUE,
controlLimit:=_StatusAi.HA, str_AIp := protections.Pgaza_na_vhode_nagnetatelia_GPA_STOP);
inits := inits + BOOL_TO_UINT(stAIp_Ini.Init);

(* Температура газа на выходе нагнетателя *)
stAIp_Ini(data_Ini := true, delay:=T#3S, inTag:=_ProtectionTags.AOS, inRunOnStart:=TRUE,
controlLimit:=_StatusAi.HA, str_AIp := protections.Pgaza_na_vyhode_nagnetatelia);
inits := inits + BOOL_TO_UINT(stAIp_Ini.Init);

(* Температура газа на выходе нагнетателя *)
stAIp_Ini(data_Ini := true, delay:=T#20S, inTag:=_ProtectionTags.AOS, inRunOnStart:=TRUE,
controlLimit:=_StatusAi.HA, str_AIp := protections.dPmaslo_gaz);
inits := inits + BOOL_TO_UINT(stAIp_Ini.Init);

(* Температура газа на выходе нагнетателя *)
stAIp_Ini(data_Ini := true, delay:=T#16S, inTag:=_ProtectionTags.AOS, inRunOnStart:=TRUE,
controlLimit:=_StatusAi.HA, str_AIp := protections.Pmaslo_sm_nizkoe);
inits := inits + BOOL_TO_UINT(stAIp_Ini.Init);

(* Температура газа на выходе нагнетателя *)
stAIp_Ini(data_Ini := true, delay:=T#16S, inTag:=_ProtectionTags.AOS, inRunOnStart:=TRUE,
controlLimit:=_StatusAi.HA, str_AIp := protections.Pmaslo_sm_vysokoe);
inits := inits + BOOL_TO_UINT(stAIp_Ini.Init);

 (* Температура газа на выходе нагнетателя *)
stAIp_Ini(data_Ini := true, delay:=T#3S, inTag:=_ProtectionTags.AOS, inRunOnStart:=TRUE,
controlLimit:=_StatusAi.HA, str_AIp := protections.Vibro_skorost_OPED_T1);
inits := inits + BOOL_TO_UINT(stAIp_Ini.Init);

 (* Температура газа на выходе нагнетателя *)
stAIp_Ini(data_Ini := true, delay:=T#3S, inTag:=_ProtectionTags.AOS, inRunOnStart:=TRUE,
controlLimit:=_StatusAi.HA, str_AIp := protections.Vibro_skorost_OPED_T2);
inits := inits + BOOL_TO_UINT(stAIp_Ini.Init);

 (* Температура газа на выходе нагнетателя *)
stAIp_Ini(data_Ini := true, delay:=T#3S, inTag:=_ProtectionTags.AOS, inRunOnStart:=TRUE,
controlLimit:=_StatusAi.HA, str_AIp := protections.Vibro_skorost_OYP_kolesa_ED_T3);
inits := inits + BOOL_TO_UINT(stAIp_Ini.Init);

 (* Температура газа на выходе нагнетателя *)
stAIp_Ini(data_Ini := true, delay:=T#3S, inTag:=_ProtectionTags.AOS, inRunOnStart:=TRUE,
controlLimit:=_StatusAi.HA, str_AIp := protections.Vibro_skorost_OP_kolesa_RH_T4);
inits := inits + BOOL_TO_UINT(stAIp_Ini.Init);

 (* Температура газа на выходе нагнетателя *)
stAIp_Ini(data_Ini := true, delay:=T#3S, inTag:=_ProtectionTags.AOS, inRunOnStart:=TRUE,
controlLimit:=_StatusAi.HA, str_AIp := protections.Vibro_skorost_OP_shesterni_RED_T5);
inits := inits + BOOL_TO_UINT(stAIp_Ini.Init);

 (* Температура газа на выходе нагнетателя *)
stAIp_Ini(data_Ini := true, delay:=T#3S, inTag:=_ProtectionTags.AOS, inRunOnStart:=TRUE,
controlLimit:=_StatusAi.HA, str_AIp := protections.Vibro_skorost_OP_shesterni_RED_T6);
inits := inits + BOOL_TO_UINT(stAIp_Ini.Init);

 (* Температура газа на выходе нагнетателя *)
stAIp_Ini(data_Ini := true, delay:=T#3S, inTag:=_ProtectionTags.AOS, inRunOnStart:=TRUE,
controlLimit:=_StatusAi.HA, str_AIp := protections.Vibro_skorost_OYP_kolesa_ED_T3);
inits := inits + BOOL_TO_UINT(stAIp_Ini.Init);

 (* Температура газа на выходе нагнетателя *)
stAIp_Ini(data_Ini := true, delay:=T#3S, inTag:=_ProtectionTags.AOS, inRunOnStart:=TRUE,
controlLimit:=_StatusAi.HA, str_AIp := protections.Vibro_skorost_OYP_kolesa_ED_T3);
inits := inits + BOOL_TO_UINT(stAIp_Ini.Init);

 (* Температура газа на выходе нагнетателя *)
stAIp_Ini(data_Ini := true, delay:=T#3S, inTag:=_ProtectionTags.AOS, inRunOnStart:=TRUE,
controlLimit:=_StatusAi.HA, str_AIp := protections.Vibro_skorost_OYP_kolesa_ED_T3);
inits := inits + BOOL_TO_UINT(stAIp_Ini.Init);

IF init THEN initiales := inits; END_IF;

(* ---- Prov_dP_mg.st ---- *)
FUNCTION_BLOCK Prov_dP_mg

VAR_IN_OUT
	StrAlg : struct_Alg;
END_VAR

VAR
	nu1Off : struct_PhaseAlgoritm;
	nu2Off : struct_PhaseAlgoritm;
	pnsOff : struct_PhaseAlgoritm;
	timer120 : struct_PhaseAlgoritm;
	dPmg_less_100 : struct_PhaseAlgoritm;
	nu1On : struct_PhaseAlgoritm;
	nu2On : struct_PhaseAlgoritm;
	pnsOn : struct_PhaseAlgoritm;
	Error_Alg : struct_PhaseAlgoritm;
	dPmg_more_100 : struct_PhaseAlgoritm;
	fb_nu1Off : fb_ph_OilPump;
	fb_nu2Off : fb_ph_OilPump;
	fb_pnsOff : fb_ph_Switch;
	fb_timer120 : fb_ph_Timer;
	fb_dPmg_less_100 : fb_ph_algoritm;
	fb_nu1On : fb_ph_OilPump;
	fb_nu2On : fb_ph_OilPump;
	fb_pnsOn : fb_ph_Switch;
	fb_Error_Alg : fb_ph_algoritm;
	fb_dPmg_more_100 : fb_ph_algoritm;
	onInit : BOOL;
END_VAR

VAR_EXTERNAL
	Im : ImConfig;
	ai : AiConfig;
END_VAR

VAR
	_sunpackerCommand : fb_sunpackerCommand;
	source : BYTE;
	cmd : BYTE;
	_statusDualInput : TYPE_statusDualInput;
	lastCmd : BYTE;
	_Answers : TYPE_Answers;
END_VAR

VAR_EXTERNAL
	ModeGpa : TYPE_ModeGpa;
	algManager : struct_AlgoritmsManager;
END_VAR

VAR
	cmd_for_Status : BYTE;
	source_for_Status : BYTE;
	command_error_for_Status : BYTE;
	resetCmdTimer : TON;
	waitReset : TON;
	resetCmdTimerPriznak : BOOL;
END_VAR

IF NOT onInit THEN
    fb_nu1Off(phaseNumber:=1, act:=_off);
    fb_nu2Off(phaseNumber:=2, act:=_off);
    fb_pnsOff(phaseNumber:=3, act:=_off);
    fb_timer120(phaseNumber:=4, delay:=T#120S);
    fb_dPmg_less_100(phaseNumber:=5);
    fb_nu1On(phaseNumber:=6, act:=_on);
    fb_nu2On(phaseNumber:=7, act:=_on);
    fb_pnsOn(phaseNumber:=8, act:=_on);
    fb_Error_Alg(phaseNumber:=9);
    fb_dPmg_more_100(phaseNumber:=10);
    onInit:=TRUE;
END_IF;

fb_nu1Off(StrPh:=nu1Off, Im:=Im.nu1);
fb_nu2Off(StrPh:=nu2Off, Im:=Im.nu2);
fb_pnsOff(StrPh:=pnsOff, Im:=Im.pns);
fb_timer120(StrPh:=timer120);
fb_dPmg_less_100(StrPh:=dPmg_less_100);
fb_nu1On(StrPh:=nu1On, Im:=Im.nu1);
fb_nu2On(StrPh:=nu2On, Im:=Im.nu2);
fb_pnsOn(StrPh:=pnsOn, Im:=Im.pns);
fb_Error_Alg(StrPh:=Error_Alg);
fb_dPmg_more_100(StrPh:=dPmg_more_100);

StrAlg.CanRun := StrAlg.inCanRun;
StrAlg.OpcCommandsDisabled := StrAlg.inOpcCommandsDisabled;

    IF StrAlg.isRuning THEN
    (* kto takoi ask
        IF	NOT nuOff.start THEN
	    NU_OFF_Ask.ask ();
    END_IF;*)

    (*
    IF	(nu_OFF_Ask.answer=Answers.ANS_YES) THEN
	    runPhase(nu1Off);
	    runPhase(nu2Off);
        runPhase(pnsOff);
	    NU_OFF_Ask.reset ();
	    runPhase(timer120);
    END_IF;*)

    (*насосы выключены - запуск проверки *)
    IF	nu1Off.top AND nu2Off.top THEN
	    runPhase(dPmg_less_100);
    END_IF;

    (*проверка перепада маслогаз по аналогу и дискрету*)
    IF	dPmg_less_100.start AND NOT dPmg_less_100.top THEN
        IF 	Im.SingleSignals.dP_maslo_gaz_Less100.Q AND ai.dPmaslo_gaz.value < 150.0 THEN
	  	    dPmg_less_100.top:=TRUE;
		    runPhase(nu1On);
            runPhase(nu2On);
            runPhase(pnsOn);
	    END_IF;
    END_IF;

    IF	Im.nu1.onStatus = _statusDualInput.STATUS_ON OR Im.nu2.onStatus = _statusDualInput.STATUS_ON  AND nu1On.start  AND nu2On.start AND NOT nu1On.top AND NOT nu2On.top THEN
	    nu1On.top := TRUE;
        nu2On.top := TRUE;
    END_IF;

    (*ошибка завершения по таймеру*)
    IF	timer120.top THEN
	    Error_Alg.ERROR := TRUE;
    ELSE
	    Error_Alg.ERROR := FALSE;
    END_IF;

    (*ыва*)
    IF	nu1On.top AND nu2On.top AND pnsOn.top THEN
	    runPhase(dPmg_more_100);
    END_IF;

    (**)
    IF	dPmg_more_100.start AND NOT dPmg_more_100.top (*AND NOT algoritms.autoNu_1.flag1 OR algoritms.autoNu_1.flag2*) THEN
	    IF 	NOT Im.SingleSignals.dP_maslo_gaz_Less100.Q AND Im.SingleSignals.dP_maslo_gaz_Less100.status = 1 AND  ai.dPmaslo_gaz.value > 150.0 THEN
    		dPmg_more_100.top :=TRUE;
		    resetPhase(timer120);
	    END_IF;
    END_IF;
END_IF;

_sunpackerCommand(command := StrAlg.inCommand);
	source := _sunpackerCommand.source;
	cmd := _sunpackerCommand.cmd;

IF cmd <> 0 AND lastCmd <> cmd AND (((NOT StrAlg.opcCommandsDisabled) AND source > 0) OR source = 0) then
	CASE BYTE_TO_INT(cmd) OF
		(*cm dRun*) 1: 	IF (StrAlg.CanRun) THEN
					StrAlg.isRuning := TRUE;
					StrAlg.isEnded := FALSE;
					StrAlg.hasError := FALSE;
					(*****************       OnRun       *****************)
                                                  algManager.nMode:=ModeGpa.MODE_PUSK_FIRST_FAZA2;

                                                  (*runPhase(timer120);
                                                  runPhase(timer5);
                                                  runPhase(Shup);
                                                  resetAiProtection(protections.dPmaslo_gaz);
                                                  resetDiProtection(protections.dPmaslo_gaz_less100);*)

					cmd_for_Status := cmd;
					source_for_Status := source;
					command_error_for_Status := 0;
				ELSE
					StrAlg.isRuning := FALSE;
					StrAlg.isEnded := FALSE;
					StrAlg.hasError := FALSE;

					cmd_for_Status := 0;
					source_for_Status := source;
					command_error_for_Status := cmd;
				END_IF;
		(*cmdReset*) 2: 	StrAlg.isRuning := FALSE;
				StrAlg.isEnded := FALSE;
				StrAlg.hasError 	:= FALSE;

                                         (*****************       OnReset       *****************)
                                        waitReset(IN:=FALSE);
                                        StrAlg.inCanRun:=FALSE;

                                        (*resetPhase(timer5);
                                        resetPhase(Shup);
                                        resetPhase(timer120);
                                        resetPhase(Net_Chast);
                                        resetPhase(mvOn);
                                        resetPhase(pGNSmore04);
                                        resetPhase(gotov_K_zagruzke);
                                        resetPhase(dPmg_Top);
                                        resetPhase(AutoPNS_Start);*)

                                        StrAlg.inOpcCommandsDisabled:=FALSE;

				cmd_for_Status := cmd;
				source_for_Status := source;
				command_error_for_Status := 0;
	END_CASE;
	resetCmdTimer(IN := false);
	resetCmdTimerPriznak := TRUE;
END_IF;
lastCmd := cmd;

resetCmdTimer(IN := resetCmdTimerPriznak, PT := T#5S);
IF resetCmdTimer.Q THEN
	resetCmdTimerPriznak := FALSE;
	source_for_Status := 0;
	cmd_for_Status := 0;
	command_error_for_Status := 0;
END_IF;

StrAlg.Start:= nu1Off.startStatus
            OR nu2Off.startStatus
            OR pnsOff.startStatus
            OR timer120.startStatus
            OR dPmg_less_100.startStatus
            OR nu1On.startStatus
            OR nu2On.startStatus
            OR pnsOn.startStatus;

StrAlg.Top := nu1Off.topStatus
            OR nu2Off.topStatus
            OR pnsOff.topStatus
            OR timer120.topStatus
            OR dPmg_less_100.topStatus
            OR nu1On.topStatus
            OR nu2On.topStatus
            OR pnsOn.topStatus;

StrAlg.Error := nu1Off.errorStatus
            OR nu2Off.errorStatus
            OR pnsOff.errorStatus
            OR timer120.errorStatus
            OR dPmg_less_100.errorStatus
            OR nu1On.errorStatus
            OR nu2On.errorStatus
            OR pnsOn.errorStatus;

(*TODO: TYPE PROGRAM CODE HERE*)
StrAlg.status :=  SHL(BYTE_TO_DWORD(source_for_Status), 29)
			OR SHL(BYTE_TO_DWORD(cmd_for_Status), 26)
			OR SHL(BYTE_TO_DWORD(command_error_for_Status), 23)
			OR SHL(BOOL_TO_DWORD(StrAlg.OpcCommandsDisabled ), 21)
			OR SHL(BOOL_TO_DWORD(StrAlg.hasError),4)
			OR SHL(BOOL_TO_DWORD(StrAlg.CanRun),2)
			OR SHL(BOOL_TO_DWORD(StrAlg.isEnded),1)
			OR BOOL_TO_DWORD(StrAlg.isRuning);

(* ---- Prov_K.st ---- *)
FUNCTION_BLOCK Prov_K

VAR_IN_OUT
	StrAlg : struct_Alg;
END_VAR

VAR
	F1_1_start : struct_PhaseAlgoritm;
	F1_2_start : struct_PhaseAlgoritm;
	F3_start : struct_PhaseAlgoritm;
	F4_Start : struct_PhaseAlgoritm;
	Start_Prov_Pusk : struct_Question;
	F4_Start_Q : struct_Question;
	fb_F1_1_start : fb_ph_algoritm;
	fb_F1_2_start : fb_ph_algoritm;
	fb_F3_start : fb_ph_algoritm;
	fb_F4_Start : fb_ph_Kran;
	algoritms : AlgoritmsConfig;
	fb_Start_Prov_Pusk : fb_Question;
	fb_F4_Start_Q : fb_Question;
	fb_kran4Open : fb_ph_Kran;
	fb_kran5Close : fb_ph_Kran;
	fb_kran4Close : fb_ph_Kran;
	fb_timer10 : fb_ph_Timer;
	fb_P_vh_vyh_more_zad : fb_ph_algoritm;
	fb_Zapoln_Norm : fb_ph_algoritm;
	fb_First_Step : fb_ph_algoritm;
	fb_Opressovka_Start : fb_Question;
	fb_PNS_NU_ON_Ask : fb_Question;
	fb_Zapolnit_kontur : fb_Question;
	onInit : BOOL;
END_VAR

VAR_EXTERNAL
	Im : ImConfig;
	ai : AiConfig;
END_VAR

VAR
	_sunpackerCommand : fb_sunpackerCommand;
	source : BYTE;
	cmd : BYTE;
	_statusDualInput : TYPE_statusDualInput;
	lastCmd : BYTE;
	_Answers : TYPE_Answers;
END_VAR

VAR_EXTERNAL
	ModeGpa : TYPE_ModeGpa;
	algManager : struct_AlgoritmsManager;
END_VAR

VAR
	cmd_for_Status : BYTE;
	source_for_Status : BYTE;
	command_error_for_Status : BYTE;
	resetCmdTimer : TON;
	waitReset : TON;
	resetCmdTimerPriznak : BOOL;
	_statusAi : TYPE_StatusAi;
	protections : ProtectionsConfig;
END_VAR

IF NOT onInit THEN
    fb_F1_1_start(phaseNumber:=1, act:=_run);
    fb_F1_2_start(phaseNumber:=2, act:=_run);
    fb_F3_start(phaseNumber:=3, act:=_run);
    fb_F4_Start(phaseNumber:=4, act:=_on);
    Start_Prov_Pusk.AnswerVariants:=_Answers.ANS_YES + _Answers.ANS_NO;
    F4_Start_Q.AnswerVariants:=_Answers.ANS_YES;
    onInit:=TRUE;
END_IF;

fb_F1_1_start(StrPh:=F1_1_start, alg := algoritms.Pusk_F_faza1);
fb_F1_2_start(StrPh:=F1_2_start, alg := algoritms.Pusk_F_faza2);
fb_F3_start(StrPh:=F3_start, alg := algoritms.Pusk_TH_faza);
fb_F4_Start(StrPh:=F4_Start, Im:=Im.Kran6);
fb_Start_Prov_Pusk(StrQ:=Start_Prov_Pusk);
fb_F4_Start_Q(StrQ:=F4_Start_Q);

StrAlg.CanRun := StrAlg.inCanRun;
StrAlg.OpcCommandsDisabled := StrAlg.inOpcCommandsDisabled;

IF StrAlg.isRuning THEN
    IF NOT F1_1_start.start THEN
	askQuestion(Start_Prov_Pusk);
    END_IF;
    IF Start_Prov_Pusk.answer = _Answers.ANS_YES THEN
	(*algoritms.F1_1.CanRun :=TRUE;*)
	runPhase(F1_1_start);
	resetQuestion(Start_Prov_Pusk);
	(*algManager.setMode(nMode:=ModeGpa.MODE_PUSKK);*)
    ELSIF	Start_Prov_Pusk.answer=_Answers.ANS_NO THEN
		resetQuestion(Start_Prov_Pusk);
		(*algoritms.F1_1.CanRun :=FALSE;*)
    END_IF;
    IF F1_1_start.top THEN
	(*algoritms.F1_2.CanRun :=TRUE;*)
	runPhase(F1_2_start);
    END_IF;
    IF 	F1_2_start.top (*AND algoritms.ppu.ppuThird*)THEN
	(*algoritms.F3.CanRun :=TRUE;*)
	runPhase(F3_start);
    END_IF;
    IF F3_start.top AND (*algoritms.ppu.ppuForth AND*) NOT F4_Start.start  THEN
	askQuestion(F4_Start_Q);
    ELSE
	resetQuestion(F4_Start_Q);
    END_IF;
    IF F4_Start_Q.answer = _Answers.ANS_YES THEN
	resetQuestion(F4_Start_Q);
	(*algoritms.F4.CanRun :=TRUE;*)
	runPhase(F4_Start);
    END_IF;
END_IF;

_sunpackerCommand(command := StrAlg.inCommand);
	source := _sunpackerCommand.source;
	cmd := _sunpackerCommand.cmd;

IF cmd <> 0 AND lastCmd <> cmd AND (((NOT StrAlg.opcCommandsDisabled) AND source > 0) OR source = 0) then
	CASE BYTE_TO_INT(cmd) OF
		(*cm dRun*) 1: 	IF (StrAlg.CanRun) THEN
					StrAlg.isRuning := TRUE;
					StrAlg.isEnded := FALSE;
					StrAlg.hasError := FALSE;
					(*****************       OnRun       *****************)
                                                  algManager.nMode:=ModeGpa.MODE_PUSK_FIRST_FAZA2;

                                                  (*runPhase(timer120);
                                                  runPhase(timer5);
                                                  runPhase(Shup);
                                                  resetAiProtection(protections.dPmaslo_gaz);
                                                  resetDiProtection(protections.dPmaslo_gaz_less100);*)

					cmd_for_Status := cmd;
					source_for_Status := source;
					command_error_for_Status := 0;
				ELSE
					StrAlg.isRuning := FALSE;
					StrAlg.isEnded := FALSE;
					StrAlg.hasError := FALSE;

					cmd_for_Status := 0;
					source_for_Status := source;
					command_error_for_Status := cmd;
				END_IF;
		(*cmdReset*) 2: 	StrAlg.isRuning := FALSE;
				StrAlg.isEnded := FALSE;
				StrAlg.hasError 	:= FALSE;

                                         (*****************       OnReset       *****************)
                                        waitReset(IN:=FALSE);
                                        StrAlg.inCanRun:=FALSE;

                                        (*resetPhase(timer5);
                                        resetPhase(Shup);
                                        resetPhase(timer120);
                                        resetPhase(Net_Chast);
                                        resetPhase(mvOn);
                                        resetPhase(pGNSmore04);
                                        resetPhase(gotov_K_zagruzke);
                                        resetPhase(dPmg_Top);
                                        resetPhase(AutoPNS_Start);*)

                                        StrAlg.inOpcCommandsDisabled:=FALSE;

				cmd_for_Status := cmd;
				source_for_Status := source;
				command_error_for_Status := 0;
	END_CASE;
	resetCmdTimer(IN := false);
	resetCmdTimerPriznak := TRUE;
END_IF;
lastCmd := cmd;

resetCmdTimer(IN := resetCmdTimerPriznak, PT := T#5S);
IF resetCmdTimer.Q THEN
	resetCmdTimerPriznak := FALSE;
	source_for_Status := 0;
	cmd_for_Status := 0;
	command_error_for_Status := 0;
END_IF;

(*StrAlg.Start:= OPC_Control.startStatus
            OR Pms_more_50.startStatus
            OR Pms_more_300.startStatus
            OR dPmg_more_100.startStatus
            OR P_zad.startStatus
            OR kran5Open.startStatus
            OR kran4Open.startStatus
            OR kran5Close.startStatus
            OR kran4Close.startStatus
            OR timer10.startStatus
            OR P_vh_vyh_more_zad.startStatus
            OR Zapoln_Norm.startStatus
            OR First_Step.startStatus;

StrAlg.Top :=  OPC_Control.topStatus
            OR Pms_more_50.topStatus
            OR Pms_more_300.topStatus
            OR dPmg_more_100.topStatus
            OR P_zad.topStatus
            OR kran5Open.topStatus
            OR kran4Open.topStatus
            OR kran5Close.topStatus
            OR kran4Close.topStatus
            OR timer10.topStatus
            OR P_vh_vyh_more_zad.topStatus
            OR Zapoln_Norm.topStatus
            OR First_Step.topStatus;

StrAlg.Error :=  OPC_Control.errorStatus
            OR Pms_more_50.errorStatus
            OR Pms_more_300.errorStatus
            OR dPmg_more_100.errorStatus
            OR P_zad.errorStatus
            OR kran5Open.errorStatus
            OR kran4Open.errorStatus
            OR kran5Close.errorStatus
            OR kran4Close.errorStatus
            OR timer10.errorStatus
            OR P_vh_vyh_more_zad.errorStatus
            OR Zapoln_Norm.errorStatus
            OR First_Step.errorStatus;*)

(*TODO: TYPE PROGRAM CODE HERE*)
StrAlg.status :=  SHL(BYTE_TO_DWORD(source_for_Status), 29)
			OR SHL(BYTE_TO_DWORD(cmd_for_Status), 26)
			OR SHL(BYTE_TO_DWORD(command_error_for_Status), 23)
			OR SHL(BOOL_TO_DWORD(StrAlg.OpcCommandsDisabled ), 21)
			OR SHL(BOOL_TO_DWORD(StrAlg.hasError),4)
			OR SHL(BOOL_TO_DWORD(StrAlg.CanRun),2)
			OR SHL(BOOL_TO_DWORD(StrAlg.isEnded),1)
			OR BOOL_TO_DWORD(StrAlg.isRuning);

(* ---- Prov_opressovka.st ---- *)
FUNCTION_BLOCK Prov_opressovka

VAR_IN_OUT
	StrAlg : struct_Alg;
END_VAR

VAR
	OPC_Control : struct_PhaseAlgoritm;
	Pms_more_50 : struct_PhaseAlgoritm;
	Pms_more_300 : struct_PhaseAlgoritm;
	dPmg_more_100 : struct_PhaseAlgoritm;
	P_zad : struct_PhaseAlgoritm;
	kran5Open : struct_PhaseAlgoritm;
	kran4Open : struct_PhaseAlgoritm;
	kran5Close : struct_PhaseAlgoritm;
	kran4Close : struct_PhaseAlgoritm;
	timer10 : struct_PhaseAlgoritm;
	P_vh_vyh_more_zad : struct_PhaseAlgoritm;
	Zapoln_Norm : struct_PhaseAlgoritm;
	First_Step : struct_PhaseAlgoritm;
	MaxZapolnenie_izm : REAL;
	Opressovka_Start : struct_Question;
	PNS_NU_ON_Ask : struct_Question;
	Zapolnit_kontur : struct_Question;
	fb_OPC_Control : fb_ph_algoritm;
	fb_Pms_more_50 : fb_ph_algoritm;
	fb_Pms_more_300 : fb_ph_algoritm;
	fb_dPmg_more_100 : fb_ph_algoritm;
	fb_P_zad : fb_ph_algoritm;
	fb_kran5Open : fb_ph_Kran;
	fb_kran4Open : fb_ph_Kran;
	fb_kran5Close : fb_ph_Kran;
	fb_kran4Close : fb_ph_Kran;
	fb_timer10 : fb_ph_Timer;
	fb_P_vh_vyh_more_zad : fb_ph_algoritm;
	fb_Zapoln_Norm : fb_ph_algoritm;
	fb_First_Step : fb_ph_algoritm;
	fb_Opressovka_Start : fb_Question;
	fb_PNS_NU_ON_Ask : fb_Question;
	fb_Zapolnit_kontur : fb_Question;
	onInit : BOOL;
END_VAR

VAR_EXTERNAL
	Im : ImConfig;
	ai : AiConfig;
END_VAR

VAR
	_sunpackerCommand : fb_sunpackerCommand;
	source : BYTE;
	cmd : BYTE;
	_statusDualInput : TYPE_statusDualInput;
	lastCmd : BYTE;
	_Answers : TYPE_Answers;
END_VAR

VAR_EXTERNAL
	ModeGpa : TYPE_ModeGpa;
	algManager : struct_AlgoritmsManager;
END_VAR

VAR
	cmd_for_Status : BYTE;
	source_for_Status : BYTE;
	command_error_for_Status : BYTE;
	resetCmdTimer : TON;
	waitReset : TON;
	resetCmdTimerPriznak : BOOL;
	_statusAi : TYPE_StatusAi;
	protections : ProtectionsConfig;
END_VAR

IF NOT onInit THEN
    fb_OPC_Control(phaseNumber:=1);
    fb_Pms_more_50(phaseNumber:=2);
    fb_Pms_more_300(phaseNumber:=3);
    fb_dPmg_more_100(phaseNumber:=4);
    fb_P_zad(phaseNumber:=5);
    fb_kran5Open(phaseNumber:=6, act:=_on);
    fb_kran4Open(phaseNumber:=7, act:=_on);
    fb_kran5Close(phaseNumber:=8, act:=_off);
    fb_kran4Close(phaseNumber:=9, act:=_off);
    fb_timer10(phaseNumber:=10, delay:=T#10S);
    fb_P_vh_vyh_more_zad(phaseNumber:=11);
    fb_Zapoln_Norm(phaseNumber:=12);
    fb_First_Step(phaseNumber:=13);
    Opressovka_Start.AnswerVariants:=_Answers.ANS_YES + _Answers.ANS_NO;
    PNS_NU_ON_Ask.AnswerVariants:=_Answers.ANS_YES;
    Zapolnit_kontur.AnswerVariants:=_Answers.ANS_YES;
    onInit:=TRUE;
END_IF;

fb_OPC_Control(StrPh:=OPC_Control);
fb_Pms_more_50(StrPh:=Pms_more_50);
fb_Pms_more_300(StrPh:=Pms_more_300);
fb_dPmg_more_100(StrPh:=dPmg_more_100);
fb_P_zad(StrPh:=P_zad);
fb_kran5Open(StrPh:=kran5Open, Im:=Im.Kran5);
fb_kran4Open(StrPh:=kran4Open, Im:=Im.Kran4);
fb_kran5Close(StrPh:=kran5Close, Im:=Im.Kran5);
fb_kran4Close(StrPh:=kran4Close, Im:=Im.Kran4);
fb_timer10(StrPh:=timer10);
fb_P_vh_vyh_more_zad(StrPh:=P_vh_vyh_more_zad);
fb_Zapoln_Norm(StrPh:=Zapoln_Norm);
fb_First_Step(StrPh:=First_Step);
fb_Opressovka_Start(StrQ:=Opressovka_Start);
fb_PNS_NU_ON_Ask(StrQ:=PNS_NU_ON_Ask);
fb_Zapolnit_kontur(StrQ:=Zapolnit_kontur);

StrAlg.CanRun := StrAlg.inCanRun;
StrAlg.OpcCommandsDisabled := StrAlg.inOpcCommandsDisabled;

IF StrAlg.isRuning THEN
   (*IF	algManager.mode <> ModeGpa.MODE_O THEN
	    askQuestion(Opressovka_Start);
    END_IF;*)

    IF	Opressovka_Start.answer=_Answers.ANS_YES THEN
	    askQuestion(Opressovka_Start);
	    Im.kran6.inOpcCommandsDisabled := FALSE;
	    (*algManager.setMode(nMode:=ModeGpa.MODE_O);*)
	    runPhase(OPC_Control);
	    resetAiProtection(protections.Pgaza_na_vyhode_nagnetatelia_GPA_STOP);
	    resetAiProtection(protections.Pgaza_na_vhode_nagnetatelia_GPA_STOP);
        ELSIF Opressovka_Start.answer=_Answers.ANS_no THEN
              resetQuestion(Opressovka_Start);
    END_IF;

    IF	OPC_Control.start AND NOT OPC_Control.top THEN
	    askQuestion(PNS_NU_ON_Ask);
    END_IF;
    IF	(PNS_NU_ON_Ask.answer=_Answers.ANS_YES) AND NOT OPC_Control.top THEN
	    OPC_Control.top:=TRUE;
	    resetQuestion(PNS_NU_ON_Ask);
    END_IF;

    IF	OPC_Control.top AND NOT Pms_more_50.start  THEN
	    Im.pns.inOpcCommandsDisabled := FALSE;
	    Im.kran6.inOpcCommandsDisabled := FALSE;
	    runPhase(Pms_more_50);
	    runPhase(Pms_more_300);
    END_IF;
    IF	OPC_Control.top AND Im.pns.onStatus = _statusDualInput.STATUS_On AND NOT dPmg_more_100.start THEN
	    Im.nu1.inOpcCommandsDisabled := FALSE;
	    Im.nu2.inOpcCommandsDisabled := FALSE;
	    runPhase(dPmg_more_100);
    END_IF;

    IF	Im.nu1.onStatus = _statusDualInput.STATUS_On OR Im.nu2.onStatus = _statusDualInput.STATUS_On AND dPmg_more_100.start AND NOT dPmg_more_100.top THEN
	    IF ai.dPmaslo_gaz.interval	>=	_statusAi.NORMAL AND
		    ai.dPmaslo_gaz.value > 150.0 AND Im.SingleSignals.dP_maslo_gaz_Less100.reliability = TRUE AND NOT Im.SingleSignals.dP_maslo_gaz_Less100.Q THEN
		    dPmg_more_100.top:=TRUE;
		    runAiProtection(protections.dPmaslo_gaz);
		    runDiProtection(protections.dPmaslo_gaz_less100);
	    END_IF;
    END_IF;

    IF	Im.pns.onStatus = _statusDualInput.STATUS_On AND Pms_more_50.start AND NOT Pms_more_50.top THEN
	        IF	ai.Pmaslo_sm_nizkoe.interval	>=	_statusAi.NORMAL AND
		        ai.Pmaslo_sm_nizkoe.value > 50.0 THEN
		        Pms_more_50.top:=TRUE;
                runAiProtection(protections.Pmaslo_sm_nizkoe);
	    END_IF;
    END_IF;

    IF	Im.pns.onStatus = _statusDualInput.STATUS_On AND Pms_more_300.start AND NOT Pms_more_300.top THEN
	    IF	ai.Pmaslo_sm_vysokoe.interval	>=	_statusAi.NORMAL AND
		    ai.Pmaslo_sm_vysokoe.value > 300.0 THEN
		    Pms_more_300.top:=TRUE;
		    runAiProtection(protections.Pmaslo_sm_vysokoe);
	    END_IF;
    END_IF;

    (*IF	dPmg_more_100.top AND Pms_more_50.top AND Pms_more_300.top THEN
	    CASE	Auto.value OF
	    0:	Im.kran3.inOpcCommandsDisabled := FALSE;
		Im.kran4.inOpcCommandsDisabled := FALSE;
		Im.kran5.inOpcCommandsDisabled := FALSE;
		Im.kran3b.inOpcCommandsDisabled := FALSE;
		resetPhase(Zapolnit_kontur);
		IF	Im.PerepadDavlenieKran1_Less100.Q THEN
			Im.kran1.inOpcCommandsDisabled := FALSE;
			Im.kran2.inOpcCommandsDisabled := FALSE;
		ELSE
			Im.kran1.inOpcCommandsDisabled := TRUE;
			Im.kran2.inOpcCommandsDisabled := TRUE;
		END_IF
		resetPhase(P_vh_vyh_more_zad);
		resetPhase(kran5Open);
		resetPhase(kran4Open);
		resetPhase(timer10);
		resetPhase(kran5Close);
		resetPhase(P_zad);
		resetPhase(First_Step);
		resetPhase(kran4Close);
		(*MaxZapolnenie_izm:=0;
		MaxZapolnenie.setValue (0);
	1:
		Zapoln_Norm.top:= MaxZapolnenie.value - MaxZapolnenie_izm > 0.4 AND MaxZapolnenie.value >= 0.4 AND MaxZapolnenie.value <= 10 AND
			ai.DGazaNaVhodeNagnetatelja.interval >= _statusAi.NORMAL AND MaxZapolnenie.value - ai.DGazaNaVhodeNagnetatelja.value > 0.4 AND
			ai.DGazaNaVyhodeNagnetatelja.interval >= _statusAi.NORMAL AND MaxZapolnenie.value - ai.DGazaNaVyhodeNagnetatelja.value > 0.4 *)
		IF	kran4Close.top AND Zapoln_Norm.top AND NOT P_zad.start THEN
			resetPhase(P_vh_vyh_more_zad);
			resetPhase(kran5Open);
			resetPhase(kran4Open);
			resetPhase(timer10);
			resetPhase(kran5Close);
			resetPhase(kran4Close);
		END_IF;
		IF	NOT kran4Close.top OR kran4Close.top AND Zapoln_Norm.top AND NOT P_zad.start THEN
		 	runPhase(P_zad);
		END_IF;
		IF NOT P_zad.top AND P_zad.start AND Zapoln_Norm.top THEN
			askQuestion(Zapolnit_kontur);
			Im.kran3.inOpcCommandsDisabled := TRUE;
			Im.kran4.inOpcCommandsDisabled := TRUE;
			Im.kran5.inOpcCommandsDisabled := TRUE;
			Im.kran3b.inOpcCommandsDisabled := TRUE;
			Im.kran1.inOpcCommandsDisabled := TRUE;
			Im.kran2.inOpcCommandsDisabled := TRUE;

		ELSIF NOT Zapoln_Norm.top AND NOT P_zad.top THEN
				resetQuestion(Zapolnit_kontur);
		END_IF;

        IF	(Zapolnit_kontur.answer=_Answers.ANS_YES) AND P_zad.start THEN
			(*MaxZapolnenie_izm:= MaxZapolnenie.value;*)
			IF 	NOT First_Step.top THEN
				runPhase(kran5Open);
			ELSE
				runPhase(kran4Open);
			END_IF;
			resetQuestion(Zapolnit_kontur);
			P_zad.top:=TRUE;
		END_IF;
                    (*

		IF	P_zad.top AND NOT kran4Close.top THEN
			MaxZapolnenie.newvalue:=MaxZapolnenie_izm;
		ELSE
			MaxZapolnenie.newvalue:= MaxZapolnenie.newvalue;
		END_IF;*)

		IF	kran5Open.top AND NOT First_Step.top THEN
			runPhase(kran4Open);
		END_IF;

        IF 	kran4Open.top AND NOT timer10.top AND NOT First_Step.top THEN
			runPhase(timer10);
		END_IF;

		IF	timer10.top AND NOT First_Step.top THEN
			runPhase(kran5Close);
		END_IF;

		IF	kran5Close.top OR First_Step.top AND kran4Open.top THEN
			runPhase(P_vh_vyh_more_zad);
        END_IF;

		IF	ai.Pgaza_na_vhode_nagnetatelia.interval >= _statusAi.NORMAL (*AND ai.Pgaza_na_vhode_nagnetatelia.value >= MaxZapolnenie.value*) AND
			ai.Pgaza_na_vyhode_nagnetatelia.interval >= _statusAi.NORMAL (*AND ai.Pgaza_na_vyhode_nagnetatelia.value >= MaxZapolnenie.value*) AND  P_vh_vyh_more_zad.start AND NOT P_vh_vyh_more_zad.top THEN
			runPhase(kran4Close);
			P_vh_vyh_more_zad.top:=TRUE;
		END_IF;

		IF	kran4Close.top THEN
			First_Step.top:=TRUE;
			Im.kran3.inOpcCommandsDisabled := FALSE;
			Im.kran4.inOpcCommandsDisabled := FALSE;
			Im.kran5.inOpcCommandsDisabled := FALSE;
			Im.kran3b.inOpcCommandsDisabled := FALSE;

            IF	Zapoln_Norm.top THEN
				resetPhase(P_zad);
			END_IF;

            IF	Im.SingleSignals.dp_kran1_Less100.Q THEN
				Im.kran1.inOpcCommandsDisabled := FALSE;
				Im.kran2.inOpcCommandsDisabled := FALSE;
			ELSE
				Im.kran1.inOpcCommandsDisabled := TRUE;
				Im.kran2.inOpcCommandsDisabled := TRUE;
			END_IF;
		ELSE
			Im.kran1.inOpcCommandsDisabled := TRUE;
			Im.kran2.inOpcCommandsDisabled := TRUE;
	    END_IF;
        END_IF;
        (*END_CASE;
END_IF;*)

_sunpackerCommand(command := StrAlg.inCommand);
	source := _sunpackerCommand.source;
	cmd := _sunpackerCommand.cmd;

IF cmd <> 0 AND lastCmd <> cmd AND (((NOT StrAlg.opcCommandsDisabled) AND source > 0) OR source = 0) then
	CASE BYTE_TO_INT(cmd) OF
		(*cm dRun*) 1: 	IF (StrAlg.CanRun) THEN
					StrAlg.isRuning := TRUE;
					StrAlg.isEnded := FALSE;
					StrAlg.hasError := FALSE;
					(*****************       OnRun       *****************)
                                                  algManager.nMode:=ModeGpa.MODE_PUSK_FIRST_FAZA2;

                                                  (*runPhase(timer120);
                                                  runPhase(timer5);
                                                  runPhase(Shup);
                                                  resetAiProtection(protections.dPmaslo_gaz);
                                                  resetDiProtection(protections.dPmaslo_gaz_less100);*)

					cmd_for_Status := cmd;
					source_for_Status := source;
					command_error_for_Status := 0;
				ELSE
					StrAlg.isRuning := FALSE;
					StrAlg.isEnded := FALSE;
					StrAlg.hasError := FALSE;

					cmd_for_Status := 0;
					source_for_Status := source;
					command_error_for_Status := cmd;
				END_IF;
		(*cmdReset*) 2: 	StrAlg.isRuning := FALSE;
				StrAlg.isEnded := FALSE;
				StrAlg.hasError 	:= FALSE;

                                         (*****************       OnReset       *****************)
                                        waitReset(IN:=FALSE);
                                        StrAlg.inCanRun:=FALSE;

                                        (*resetPhase(timer5);
                                        resetPhase(Shup);
                                        resetPhase(timer120);
                                        resetPhase(Net_Chast);
                                        resetPhase(mvOn);
                                        resetPhase(pGNSmore04);
                                        resetPhase(gotov_K_zagruzke);
                                        resetPhase(dPmg_Top);
                                        resetPhase(AutoPNS_Start);*)

                                        StrAlg.inOpcCommandsDisabled:=FALSE;

				cmd_for_Status := cmd;
				source_for_Status := source;
				command_error_for_Status := 0;
	END_CASE;
	resetCmdTimer(IN := false);
	resetCmdTimerPriznak := TRUE;
END_IF;
lastCmd := cmd;

resetCmdTimer(IN := resetCmdTimerPriznak, PT := T#5S);
IF resetCmdTimer.Q THEN
	resetCmdTimerPriznak := FALSE;
	source_for_Status := 0;
	cmd_for_Status := 0;
	command_error_for_Status := 0;
END_IF;

StrAlg.Start:= OPC_Control.startStatus
            OR Pms_more_50.startStatus
            OR Pms_more_300.startStatus
            OR dPmg_more_100.startStatus
            OR P_zad.startStatus
            OR kran5Open.startStatus
            OR kran4Open.startStatus
            OR kran5Close.startStatus
            OR kran4Close.startStatus
            OR timer10.startStatus
            OR P_vh_vyh_more_zad.startStatus
            OR Zapoln_Norm.startStatus
            OR First_Step.startStatus;

StrAlg.Top :=  OPC_Control.topStatus
            OR Pms_more_50.topStatus
            OR Pms_more_300.topStatus
            OR dPmg_more_100.topStatus
            OR P_zad.topStatus
            OR kran5Open.topStatus
            OR kran4Open.topStatus
            OR kran5Close.topStatus
            OR kran4Close.topStatus
            OR timer10.topStatus
            OR P_vh_vyh_more_zad.topStatus
            OR Zapoln_Norm.topStatus
            OR First_Step.topStatus;

StrAlg.Error :=  OPC_Control.errorStatus
            OR Pms_more_50.errorStatus
            OR Pms_more_300.errorStatus
            OR dPmg_more_100.errorStatus
            OR P_zad.errorStatus
            OR kran5Open.errorStatus
            OR kran4Open.errorStatus
            OR kran5Close.errorStatus
            OR kran4Close.errorStatus
            OR timer10.errorStatus
            OR P_vh_vyh_more_zad.errorStatus
            OR Zapoln_Norm.errorStatus
            OR First_Step.errorStatus;

(*TODO: TYPE PROGRAM CODE HERE*)
StrAlg.status :=  SHL(BYTE_TO_DWORD(source_for_Status), 29)
			OR SHL(BYTE_TO_DWORD(cmd_for_Status), 26)
			OR SHL(BYTE_TO_DWORD(command_error_for_Status), 23)
			OR SHL(BOOL_TO_DWORD(StrAlg.OpcCommandsDisabled ), 21)
			OR SHL(BOOL_TO_DWORD(StrAlg.hasError),4)
			OR SHL(BOOL_TO_DWORD(StrAlg.CanRun),2)
			OR SHL(BOOL_TO_DWORD(StrAlg.isEnded),1)
			OR BOOL_TO_DWORD(StrAlg.isRuning);

(* ---- Prov_PMS.st ---- *)
FUNCTION_BLOCK Prov_PMS

VAR_IN_OUT
	StrAlg : struct_Alg;
END_VAR

VAR
	pnsOff : struct_PhaseAlgoritm;
	timer120 : struct_PhaseAlgoritm;
	Pms_less_25 : struct_PhaseAlgoritm;
	Pms_less_250 : struct_PhaseAlgoritm;
	Error_Alg : struct_PhaseAlgoritm;
	fb_Pms_less_25 : fb_ph_algoritm;
	fb_Pms_less_250 : fb_ph_algoritm;
	fb_pnsOff : fb_ph_Switch;
	fb_timer120 : fb_ph_Timer;
	fb_Error_Alg : fb_ph_algoritm;
	onInit : BOOL;
END_VAR

VAR_EXTERNAL
	Im : ImConfig;
	ai : AiConfig;
END_VAR

VAR
	_sunpackerCommand : fb_sunpackerCommand;
	source : BYTE;
	cmd : BYTE;
	_statusDualInput : TYPE_statusDualInput;
	lastCmd : BYTE;
	_Answers : TYPE_Answers;
END_VAR

VAR_EXTERNAL
	ModeGpa : TYPE_ModeGpa;
	algManager : struct_AlgoritmsManager;
END_VAR

VAR
	cmd_for_Status : BYTE;
	source_for_Status : BYTE;
	command_error_for_Status : BYTE;
	resetCmdTimer : TON;
	waitReset : TON;
	resetCmdTimerPriznak : BOOL;
	_statusAi : TYPE_StatusAi;
END_VAR

IF NOT onInit THEN
    fb_pnsOff(phaseNumber:=1, act:=_off);
    fb_timer120(phaseNumber:=2, delay:=T#120S);
    fb_Pms_less_25(phaseNumber:=3);
    fb_Pms_less_250(phaseNumber:=4);
    fb_Error_Alg(phaseNumber:=5);
    onInit:=TRUE;
END_IF;

fb_pnsOff(StrPh:=pnsOff, Im:=Im.pns);
fb_timer120(StrPh:=timer120);
fb_Pms_less_25(StrPh:=Pms_less_25);
fb_Pms_less_250(StrPh:=Pms_less_250);
fb_Error_Alg(StrPh:=Error_Alg);

StrAlg.CanRun := StrAlg.inCanRun;
StrAlg.OpcCommandsDisabled := StrAlg.inOpcCommandsDisabled;

IF StrAlg.isRuning THEN
   (*IF NOT pnsOff.start THEN
	    PNS_OFF_Ask.ask ();
    END_IF;
    IF	(PNS_OFF_Ask.answer=Answers.ANS_YES) THEN
	    runPhase(pnsOff);
        PNS_OFF_Ask.reset ();
	    IF NOT (Pms_less_250.top AND Pms_less_25.top) THEN
	    	runPhase(timer120);
	    END_IF;
    END_IF;*)

    (*запуск проверок давления*)
    IF	pnsOff.top  THEN
        runPhase(Pms_less_25);
	    runPhase(Pms_less_250);
    END_IF;

    (*проверка давления масла низкое*)
    IF	Pms_less_25.start AND NOT Pms_less_25.top THEN
	    IF 	ai.Pmaslo_sm_nizkoe.interval>=_statusAi.NORMAL AND ai.Pmaslo_sm_nizkoe.value < 25.0 THEN
	  	    Pms_less_25.top:=TRUE;
	    END_IF;
    END_IF;

    IF	Pms_less_250.start AND NOT Pms_less_250.top THEN
	    IF	ai.Pmaslo_sm_vysokoe.interval>=_statusAi.NORMAL AND ai.Pmaslo_sm_vysokoe.value < 250.0 THEN
	  	    Pms_less_250.top:=TRUE;
	    END_IF;
    END_IF;

    (*ошибка заврешия алгоритма по таймеру*)
    IF	timer120.top THEN
	    Error_Alg.ERROR := TRUE;
    ELSE
	    Error_Alg.ERROR := FALSE;
    END_IF;

    (*если проверка прошла - сброс таймера *)
    IF	Pms_less_250.top AND Pms_less_25.top  THEN
        resetPhase(timer120);
    END_IF;
END_IF;

_sunpackerCommand(command := StrAlg.inCommand);
	source := _sunpackerCommand.source;
	cmd := _sunpackerCommand.cmd;

IF cmd <> 0 AND lastCmd <> cmd AND (((NOT StrAlg.opcCommandsDisabled) AND source > 0) OR source = 0) then
	CASE BYTE_TO_INT(cmd) OF
		(*cm dRun*) 1: 	IF (StrAlg.CanRun) THEN
					StrAlg.isRuning := TRUE;
					StrAlg.isEnded := FALSE;
					StrAlg.hasError := FALSE;
					(*****************       OnRun       *****************)
                                                  algManager.nMode:=ModeGpa.MODE_PUSK_FIRST_FAZA2;

                                                  (*runPhase(timer120);
                                                  runPhase(timer5);
                                                  runPhase(Shup);
                                                  resetAiProtection(protections.dPmaslo_gaz);
                                                  resetDiProtection(protections.dPmaslo_gaz_less100);*)

					cmd_for_Status := cmd;
					source_for_Status := source;
					command_error_for_Status := 0;
				ELSE
					StrAlg.isRuning := FALSE;
					StrAlg.isEnded := FALSE;
					StrAlg.hasError := FALSE;

					cmd_for_Status := 0;
					source_for_Status := source;
					command_error_for_Status := cmd;
				END_IF;
		(*cmdReset*) 2: 	StrAlg.isRuning := FALSE;
				StrAlg.isEnded := FALSE;
				StrAlg.hasError 	:= FALSE;

                                         (*****************       OnReset       *****************)
                                        waitReset(IN:=FALSE);
                                        StrAlg.inCanRun:=FALSE;

                                        (*resetPhase(timer5);
                                        resetPhase(Shup);
                                        resetPhase(timer120);
                                        resetPhase(Net_Chast);
                                        resetPhase(mvOn);
                                        resetPhase(pGNSmore04);
                                        resetPhase(gotov_K_zagruzke);
                                        resetPhase(dPmg_Top);
                                        resetPhase(AutoPNS_Start);*)

                                        StrAlg.inOpcCommandsDisabled:=FALSE;

				cmd_for_Status := cmd;
				source_for_Status := source;
				command_error_for_Status := 0;
	END_CASE;
	resetCmdTimer(IN := false);
	resetCmdTimerPriznak := TRUE;
END_IF;
lastCmd := cmd;

resetCmdTimer(IN := resetCmdTimerPriznak, PT := T#5S);
IF resetCmdTimer.Q THEN
	resetCmdTimerPriznak := FALSE;
	source_for_Status := 0;
	cmd_for_Status := 0;
	command_error_for_Status := 0;
END_IF;

StrAlg.Start:= pnsOff.startStatus
            OR timer120.startStatus
            OR Pms_less_25.startStatus
            OR Pms_less_250.startStatus;

StrAlg.Top :=  pnsOff.topStatus
            OR timer120.topStatus
            OR Pms_less_25.topStatus
            OR Pms_less_250.topStatus;

StrAlg.Error :=  pnsOff.errorStatus
            OR timer120.errorStatus
            OR Pms_less_25.errorStatus
            OR Pms_less_250.errorStatus;

(*TODO: TYPE PROGRAM CODE HERE*)
StrAlg.status :=  SHL(BYTE_TO_DWORD(source_for_Status), 29)
			OR SHL(BYTE_TO_DWORD(cmd_for_Status), 26)
			OR SHL(BYTE_TO_DWORD(command_error_for_Status), 23)
			OR SHL(BOOL_TO_DWORD(StrAlg.OpcCommandsDisabled ), 21)
			OR SHL(BOOL_TO_DWORD(StrAlg.hasError),4)
			OR SHL(BOOL_TO_DWORD(StrAlg.CanRun),2)
			OR SHL(BOOL_TO_DWORD(StrAlg.isEnded),1)
			OR BOOL_TO_DWORD(StrAlg.isRuning);

(* ---- Pusk_first_faza1.st ---- *)
FUNCTION_BLOCK Pusk_first_faza1

VAR_IN_OUT
	StrAlg : struct_Alg;
END_VAR

VAR
	timer240 : struct_PhaseAlgoritm;
	pmsMore50 : struct_PhaseAlgoritm;
	pnsOn : struct_PhaseAlgoritm;
	pmsMore300 : struct_PhaseAlgoritm;
	Protection_Pms : struct_PhaseAlgoritm;
	Error_Alg : struct_PhaseAlgoritm;
	fb_timer240 : fb_ph_Timer;
	fb_PnmMore50 : fb_ph_algoritm;
	fb_PnsOn : fb_ph_Switch;
	fb_PmsMore300 : fb_ph_algoritm;
	fb_Protection_Pms : fb_ph_algoritm;
	fb_Error_Alg : fb_ph_algoritm;
	_sunpackerCommand : fb_sunpackerCommand;
	_PhaseAlgoritmAction : TYPE_PhaseAlgoritmAction;
	_statusDualInput : TYPE_statusDualInput;
	_Answers : TYPE_Answers;
	source : BYTE;
	cmd : BYTE;
	lastCmd : BYTE;
	source_for_Status : BYTE;
	cmd_for_Status : BYTE;
	command_error_for_Status : BYTE;
	resetCmdTimer : TON;
	resetCmdTimerPriznak : BOOL;
	onInit : BOOL;
	waitReset : TON;
END_VAR

VAR_EXTERNAL
	ModeGpa : TYPE_ModeGpa;
	algManager : struct_AlgoritmsManager;
	IM : ImConfig;
	protections : ProtectionsConfig;
END_VAR

VAR
	_statusAi : TYPE_StatusAi;
END_VAR

VAR_EXTERNAL
	ai : AiConfig;
END_VAR

IF NOT onInit THEN

         fb_timer240(phaseNumber:=0, delay:=T#240S);
         fb_PnmMore50(phaseNumber:=1);
         fb_PnsOn(phaseNumber:=2, act:=_on);
         fb_PmsMore300(phaseNumber:=3);
         fb_Protection_Pms(phaseNumber:=4);
         fb_Error_Alg(phaseNumber:=5);

onInit:=TRUE;
END_IF;

fb_timer240(StrPh:=timer240);
fb_PnmMore50(StrPh:=pmsMore50);
fb_PnsOn(StrPh:=pnsOn, IM := Im.pns);
fb_PmsMore300(StrPh:=pmsMore300);
fb_Protection_Pms(StrPh:=Protection_Pms);
fb_Error_Alg(StrPh:=Error_Alg);

StrAlg.CanRun := StrAlg.inCanRun;
StrAlg.OpcCommandsDisabled := StrAlg.inOpcCommandsDisabled;

IF StrAlg.isRuning THEN

    StrAlg.hasError := pnsOn.error;

    (* не взведены защиты - запуск таймера *)
    IF NOT Protection_Pms.top THEN
	runPhase(timer240);
    END_IF;

    (* не начался запуск пнс - запуск пнс *)
    IF NOT pnsOn.start THEN
	runPhase(pnsOn);
    END_IF;

    (* запуск пнс завершен - запус защит *)
    IF pnsOn.top THEN
         runPhase(pmsMore50);
         runPhase(pmsMore300);
    END_IF;

    (* не завершился запуск защиты 50 - проверка давления 50 *)
    IF pmsMore50.start AND (NOT pmsMore50.top) THEN
	IF ai.Pmaslo_sm_nizkoe.interval = _statusAi.NORMAL AND ai.Pmaslo_sm_nizkoe.value > 50.0  THEN
	   pmsMore50.top := TRUE;
          END_IF;
    END_IF;

    (* не завершился запуск защиты 300 - проверка давления 300 *)
    IF  pmsMore300.start AND (NOT pmsMore300.top) THEN
	IF ai.Pmaslo_sm_vysokoe.interval = _statusAi.NORMAL AND ai.Pmaslo_sm_vysokoe.value > 300.0  THEN
	    pmsMore300.top := TRUE;
	END_IF;
    END_IF;

    (* давление было проверено - запуск защит *)
    IF pmsMore50.top AND pmsMore300.top THEN
        runPhase(Protection_Pms);
    END_IF;

    (* запуск защит не завршен - запуск защит *)
    IF Protection_Pms.start AND (NOT Protection_Pms.top) THEN
	runAiProtection(protections.Pmaslo_sm_nizkoe);
          runAiProtection(protections.Pmaslo_sm_vysokoe);
          Protection_Pms.top := TRUE;
    END_IF;

    (* таймер завершился до запуска защит - ошибка *)
    IF timer240.top THEN
        Error_Alg.ERROR := TRUE; (*не понятное куда его сунуть и нужен ли он*)
    ELSE
        Error_Alg.ERROR := FALSE;
    END_IF;

    (* защиты выствалены до завршения таймера - сброс таймера *)
    IF Protection_Pms.top THEN
	resetPhase(timer240);
    END_IF;

    StrAlg.isEnded:= pnsOn.Top AND Protection_Pms.Top (*Как будто нужно таймер *);
END_IF;

StrAlg.CanRun := StrAlg.inCanRun;
StrAlg.OpcCommandsDisabled := StrAlg.inOpcCommandsDisabled;

(* ---- Если управление с ВУ заблокировано, то  передаем команду из алгоритма ---- *)
IF StrAlg.inOpcCommandsDisabled THEN
	StrAlg.inCommand := StrAlg.inCommand_Alg;
ELSE (* иначе передаем команду с АРМа*)
	StrAlg.inCommand := StrAlg.inCommand_ARM;
END_IF;

_sunpackerCommand(command := StrAlg.inCommand);
	source := _sunpackerCommand.source;
	cmd := _sunpackerCommand.cmd;

IF cmd <> 0 AND lastCmd <> cmd AND (((NOT StrAlg.opcCommandsDisabled) AND source > 0) OR source = 0) then
	CASE BYTE_TO_INT(cmd) OF
		(*cmdRun*) 1: 	IF (StrAlg.CanRun) THEN
					StrAlg.isRuning := TRUE;
					StrAlg.isEnded := FALSE;
					StrAlg.hasError := FALSE;
					(*****************       OnRun       *****************)
                                                  algManager.nMode:=ModeGpa.MODE_PUSK_FIRST_FAZA1;

                                                  runPhase(pnsOn);
                                                  resetAiProtection(protections.Pmaslo_sm_nizkoe);
                                                  resetAiProtection(protections.Pmaslo_sm_vysokoe);

					cmd_for_Status := cmd;
					source_for_Status := source;
					command_error_for_Status := 0;
				ELSE
					StrAlg.isRuning := FALSE;
					StrAlg.isEnded := FALSE;
					StrAlg.hasError := FALSE;

					cmd_for_Status := 0;
					source_for_Status := source;
					command_error_for_Status := cmd;
				END_IF;
		(*cmdReset*) 2: 	StrAlg.isRuning := FALSE;
				StrAlg.isEnded := FALSE;
				StrAlg.hasError 	:= FALSE;

                                         (*****************       OnReset       *****************)
                                        waitReset(IN:=FALSE);
                                        StrAlg.inCanRun:=FALSE;

                                        resetPhase(timer240);
                                        resetPhase(pmsMore50);
                                        resetPhase(pnsOn);
                                        resetPhase(pmsMore300);
                                        resetPhase(Protection_Pms);
                                        resetPhase(Error_Alg);

                                        StrAlg.inOpcCommandsDisabled:=FALSE;

				cmd_for_Status := cmd;
				source_for_Status := source;
				command_error_for_Status := 0;
	END_CASE;
	resetCmdTimer(IN := false);
	resetCmdTimerPriznak := TRUE;
END_IF;
lastCmd := cmd;

resetCmdTimer(IN := resetCmdTimerPriznak, PT := T#5S);
IF resetCmdTimer.Q THEN
	resetCmdTimerPriznak := FALSE;
	source_for_Status := 0;
	cmd_for_Status := 0;
	command_error_for_Status := 0;
END_IF;

StrAlg.Start:= timer240.startStatus
            OR pmsMore50.startStatus
            OR pnsOn.startStatus
            OR Error_Alg.startStatus
            OR pmsMore300.startStatus
            OR Protection_Pms.startStatus;

StrAlg.Error := timer240.errorStatus
            OR pmsMore50.errorStatus
            OR pnsOn.errorStatus
            OR Error_Alg.errorStatus
            OR pmsMore300.errorStatus
            OR Protection_Pms.errorStatus;

StrAlg.Top := timer240.topStatus
            OR pmsMore50.topStatus
            OR pnsOn.topStatus
            OR Error_Alg.topStatus
            OR pmsMore300.topStatus
            OR Protection_Pms.topStatus;

(*TODO: TYPE PROGRAM CODE HERE*)
StrAlg.status :=  SHL(BYTE_TO_DWORD(source_for_Status), 29)
			OR SHL(BYTE_TO_DWORD(cmd_for_Status), 26)
			OR SHL(BYTE_TO_DWORD(command_error_for_Status), 23)
			OR SHL(BOOL_TO_DWORD(StrAlg.OpcCommandsDisabled ), 21)
			OR SHL(BOOL_TO_DWORD(StrAlg.hasError),4)
			OR SHL(BOOL_TO_DWORD(StrAlg.CanRun),2)
			OR SHL(BOOL_TO_DWORD(StrAlg.isEnded),1)
			OR BOOL_TO_DWORD(StrAlg.isRuning);

(* ---- Pusk_first_faza2.st ---- *)
FUNCTION_BLOCK Pusk_first_faza2

VAR_IN_OUT
	StrAlg : struct_Alg;
END_VAR

VAR
	nu1On : struct_PhaseAlgoritm;
	nu2On : struct_PhaseAlgoritm;
	timer240 : struct_PhaseAlgoritm;
	dPmg_more100 : struct_PhaseAlgoritm;
	Auto_NU1 : struct_PhaseAlgoritm;
	Error_Alg : struct_PhaseAlgoritm;
	fb_timer240 : fb_ph_Timer;
	fb_nu1On : fb_ph_OilPump;
	fb_nu2On : fb_ph_OilPump;
	fb_dPmg_more100 : fb_ph_algoritm;
	fb_Auto_NU1 : fb_ph_algoritm;
	fb_Error_Alg : fb_ph_algoritm;
	_sunpackerCommand : fb_sunpackerCommand;
	_statusDualInput : TYPE_statusDualInput;
	_Answers : TYPE_Answers;
	source : BYTE;
	cmd : BYTE;
	lastCmd : BYTE;
	source_for_Status : BYTE;
	cmd_for_Status : BYTE;
	command_error_for_Status : BYTE;
	resetCmdTimer : TON;
	resetCmdTimerPriznak : BOOL;
	onInit : BOOL;
	waitReset : TON;
END_VAR

VAR_EXTERNAL
	ModeGpa : TYPE_ModeGpa;
	algManager : struct_AlgoritmsManager;
	IM : ImConfig;
	protections : ProtectionsConfig;
	algoritms : AlgoritmsConfig;
	ai : AiConfig;
END_VAR

VAR
	statusAi : TYPE_StatusAi;
END_VAR

IF NOT onInit THEN
         fb_nu1On(phaseNumber:=1, act:=_on );
         fb_nu2On(phaseNumber:=2, act:=_on);
         fb_dPmg_more100(phaseNumber:=3);
         fb_Error_Alg(phaseNumber:=4);
         fb_Auto_NU1(phaseNumber:=5);
onInit:=TRUE;
END_IF;

fb_timer240(StrPh:=timer240);
fb_nu1On(StrPh:= nu1On,Im:=Im.nu1);
fb_nu2On(StrPh:= nu2On,Im:=Im.nu2);
fb_dPmg_more100(StrPh:=dPmg_more100);
fb_Auto_NU1(StrPh:=Auto_NU1, alg:=algoritms.autoNu); (*komu ono nujno to blat *)
fb_Error_Alg(StrPh:=Error_Alg);

StrAlg.CanRun := StrAlg.inCanRun;
StrAlg.OpcCommandsDisabled := StrAlg.inOpcCommandsDisabled;

IF StrAlg.isRuning THEN

    StrAlg.hasError := nu1On.error AND nu2On.error AND Auto_NU1.error;

    (* защита не возведена - запускаем таймер *)
    IF NOT dPmg_more100.top THEN
	runPhase(timer240);
    END_IF;

    (* носос 1 не включен - включаем насос*)
    IF NOT nu1On.start THEN
	runPhase(nu1On);
    END_IF;

    (* носос 2 не включен - включаем насос*)
    IF NOT nu2On.start THEN
	runPhase(nu2On);
    END_IF;

    (* один из насосов включен - включение защиты *)
    IF ((IM.nu1.onStatus = _statusDualInput.status_on OR IM.nu2.onStatus = _statusDualInput.status_on) AND  (nu1On.start OR nu2On.Start)) THEN
	runPhase(dPmg_more100);
	nu1On.top:=TRUE;
          nu2On.top:=TRUE;
    END_IF;

    (* фаза защиты активна - включение защиты *)
    IF dPmg_more100.start AND NOT dPmg_more100.top THEN
	IF NOT IM.SingleSignals.dP_maslo_gaz_Less100.Q AND IM.SingleSignals.dP_maslo_gaz_Less100.status = 1 AND
	ai.dPmaslo_gaz.interval >= statusAi.normal AND ai.dPmaslo_gaz.value > 150.0 THEN
              dPmg_more100.top:=TRUE;
	END_IF;
    END_IF;

    (*таймер завершился до возведения защит - ошибка *)
    IF timer240.top THEN
	Error_Alg.error := TRUE;
    ELSE
	Error_Alg.error := FALSE;
    END_IF;

    IF dPmg_more100.top AND nu1On.top AND nu2On.top THEN
	Auto_NU1.top:=TRUE;
	runAiProtection(protections.dPmaslo_gaz);
          runDiProtection(protections.dPmaslo_gaz_less100);
	resetAiProtection(protections.Pgaza_na_vhode_nagnetatelia_GPA_STOP);
	resetAiProtection(protections.Pgaza_na_vyhode_nagnetatelia_GPA_STOP);
	algoritms.autoNu.CanRun:=TRUE;
	(*algoritms.autoNu.run ();ниче не ясно*)
	resetPhase(timer240);
    END_IF;
END_IF;

StrAlg.CanRun := StrAlg.inCanRun;
StrAlg.OpcCommandsDisabled := StrAlg.inOpcCommandsDisabled;

(* ---- Если управление с ВУ заблокировано, то  передаем команду из алгоритма ---- *)
IF StrAlg.inOpcCommandsDisabled THEN
	StrAlg.inCommand := StrAlg.inCommand_Alg;
ELSE (* иначе передаем команду с АРМа*)
	StrAlg.inCommand := StrAlg.inCommand_ARM;
END_IF;

_sunpackerCommand(command := StrAlg.inCommand);
	source := _sunpackerCommand.source;
	cmd := _sunpackerCommand.cmd;

IF cmd <> 0 AND lastCmd <> cmd AND (((NOT StrAlg.opcCommandsDisabled) AND source > 0) OR source = 0) then
	CASE BYTE_TO_INT(cmd) OF
		(*cmdRun*) 1: 	IF (StrAlg.CanRun) THEN
					StrAlg.isRuning := TRUE;
					StrAlg.isEnded := FALSE;
					StrAlg.hasError := FALSE;
					(*****************       OnRun       *****************)
                                                  algManager.nMode:=ModeGpa.MODE_PUSK_FIRST_FAZA2;

                                                  runPhase(timer240);
                                                  runPhase(nu1On);
                                                  runPhase(nu2On);
                                                  resetAiProtection(protections.dPmaslo_gaz);
                                                  resetDiProtection(protections.dPmaslo_gaz_less100);

					cmd_for_Status := cmd;
					source_for_Status := source;
					command_error_for_Status := 0;
				ELSE
					StrAlg.isRuning := FALSE;
					StrAlg.isEnded := FALSE;
					StrAlg.hasError := FALSE;

					cmd_for_Status := 0;
					source_for_Status := source;
					command_error_for_Status := cmd;
				END_IF;
		(*cmdReset*) 2: 	StrAlg.isRuning := FALSE;
				StrAlg.isEnded := FALSE;
				StrAlg.hasError 	:= FALSE;

                                         (*****************       OnReset       *****************)
                                        waitReset(IN:=FALSE);
                                        StrAlg.inCanRun:=FALSE;

                                        resetPhase(nu1On);
                                        resetPhase(nu2On);
                                        resetPhase(timer240);
                                        resetPhase(dPmg_more100);
                                        resetPhase(Auto_NU1);
                                        resetPhase(Error_Alg);

                                        StrAlg.inOpcCommandsDisabled:=FALSE;

				cmd_for_Status := cmd;
				source_for_Status := source;
				command_error_for_Status := 0;
	END_CASE;
	resetCmdTimer(IN := false);
	resetCmdTimerPriznak := TRUE;
END_IF;
lastCmd := cmd;

resetCmdTimer(IN := resetCmdTimerPriznak, PT := T#5S);
IF resetCmdTimer.Q THEN
	resetCmdTimerPriznak := FALSE;
	source_for_Status := 0;
	cmd_for_Status := 0;
	command_error_for_Status := 0;
END_IF;

StrAlg.Start:= timer240.startStatus
            OR nu1On.startStatus
            OR nu2On.startStatus
            OR dPmg_more100.startStatus
            OR Auto_NU1.startStatus
            OR Error_Alg.startStatus;

StrAlg.Error := timer240.errorStatus
            OR nu1On.errorStatus
            OR nu2On.errorStatus
            OR dPmg_more100.errorStatus
            OR Auto_NU1.errorStatus
            OR Error_Alg.errorStatus;

StrAlg.Top := timer240.topStatus
            OR nu1On.topStatus
            OR nu2On.topStatus
            OR dPmg_more100.topStatus
            OR Auto_NU1.topStatus
            OR Error_Alg.topStatus;

(*TODO: TYPE PROGRAM CODE HERE*)
StrAlg.status :=  SHL(BYTE_TO_DWORD(source_for_Status), 29)
			OR SHL(BYTE_TO_DWORD(cmd_for_Status), 26)
			OR SHL(BYTE_TO_DWORD(command_error_for_Status), 23)
			OR SHL(BOOL_TO_DWORD(StrAlg.OpcCommandsDisabled ), 21)
			OR SHL(BOOL_TO_DWORD(StrAlg.hasError),4)
			OR SHL(BOOL_TO_DWORD(StrAlg.CanRun),2)
			OR SHL(BOOL_TO_DWORD(StrAlg.isEnded),1)
			OR BOOL_TO_DWORD(StrAlg.isRuning);
